// TIA Portal project "Project2" (V20)

(* hardware
DEVICE "S7-1200 station_1"  S7-1200 Station
   slot 0: "Rack_0"  S7-1200 Rack  Rack  V1.0
   slot 1: "PLC_1"  CPU 1214C DC/DC/DC  6ES7 214-1AG40-0XB0  V4.5
*)

// ===== PLC "PLC_1"  CPU 1214C DC/DC/DC =====

VAR_GLOBAL   // PLC tag table "Default tag table"
   "Axis_2_Pulse" AT %Q0.1 : Bool;
   "Axis_1_Direction" AT %Q0.6 : Bool;
   "Axis_Conveyor" AT %Q0.3 : Bool;
   "Axis_1_Pulse" AT %Q0.2 : Bool;
   "Axis_2_Direction" AT %Q0.4 : Bool;
   "M_Emergency" AT %M0.1 : Bool;
   "Velocity_1" AT %MD54 : Real;
   "Velocity_2" AT %MD58 : Real;
   "Velocity_3" AT %MD62 : Real;
   "I_Start" AT %I0.5 : Bool;
   "Set Velocity Conveyor" AT %MD80 : Real;
   "Velocity Conveyor" AT %MD84 : Real;
   "DeltaX_JobRev" AT %M200.1 : Bool;
   "DeltaX_JobFwd" AT %M200.0 : Bool;
   "DeltaX_Auto" AT %M11.0 : Bool;
   "EXC_Absolute" AT %M10.2 : Bool;
   "Po.S Done" AT %M120.0 : Bool;
   "Pos.DoneP" AT %M120.1 : Bool;
   "Servo#01 Fwd" AT %M2.0 : Bool;
   "Servo#02 Rev" AT %M2.1 : Bool;
   "Servo#02 Fwd" AT %M2.2 : Bool;
   "Servo#01 Rev" AT %M2.3 : Bool;
   "Servo#03 Fwd" AT %M2.4 : Bool;
   "Servo#03 Rev" AT %M2.5 : Bool;
   "Axis X_Work Complete" AT %M40.0 : Bool;
   "Axis Y_Work Complete" AT %M40.1 : Bool;
   "Axis Z_Work Complete" AT %M40.2 : Bool;
   "Axis X Busy" AT %M40.4 : Bool;
   "Axis Y Busy" AT %M40.5 : Bool;
   "Axis Z Busy" AT %M40.6 : Bool;
   "DeltaX_No Movement" AT %M40.7 : Bool;
   "I_Emergency" AT %I0.4 : Bool;
   "Vacum" AT %Q0.7 : Bool;
   "I_switch_1" AT %I0.0 : Bool;
   "DeltaX_Hbusy" AT %M111.0 : Bool;
   "DeltaX_Home" AT %M110.0 : Bool;
   "DeltaX_Start Home" AT %M110.1 : Bool;
   "tag_35" AT %M1000.0 : Bool;
   "I_switch_2" AT %I0.1 : Bool;
   "DeltaX1_1_Hbusy" AT %M111.1 : Bool;
   "Tag_39" AT %M1001.0 : Bool;
   "DeltaX2_Hbusy" AT %M111.2 : Bool;
   "DeltaX2_1_Hbusy" AT %M111.3 : Bool;
   "I_switch_3" AT %I0.2 : Bool;
   "Tag_40" AT %M1002.0 : Bool;
   "DeltaX3.1_Hbusy" AT %M111.5 : Bool;
   "DeltaX3_Hbusy" AT %M111.4 : Bool;
   "DeltaX_Home Busy" AT %M111.6 : Bool;
   "Home rest" AT %M110.2 : Bool;
   "EXC_Home P" AT %M152.0 : Bool;
   "Tag_28" AT %M305.1 : Bool;
   "ExC Home" AT %M150.7 : Bool;
   "Tag_27" AT %M305.0 : Bool;
   "Done_Home" AT %M10.3 : Bool;
   "Provess Data" AT %MW78 : Int;
   "Q_Reset_lamp" AT %Q8.5 : Bool;
   "PosionX_C#" AT %MD440 : Real;
   "PosionY_C#" AT %MD444 : Real;
   "Velocity_angular" AT %MD550 : Real;
   "DeltaX_Stop" AT %M11.1 : Bool;
   "bt_autoc#" AT %M110.3 : Bool;
   "bt_StopC#" AT %M110.4 : Bool;
   "DeltaX_Vacuum" AT %M153.0 : Bool;
   "Start Process" AT %M30.1 : Bool;
   "DeltaX_start Process" AT %M12.0 : Bool;
   "DeltaX_C# Enable" AT %M30.2 : Bool;
   "Tag_36" AT %M30.3 : Bool;
   "Step 7 ExC" AT %M151.1 : Bool;
   "Enable Scan" AT %M999.1 : Bool;
   "Tag_44" AT %M302.1 : Bool;
   "Tag_1" AT %M999.0 : Bool;
   "Step 1 Exc" AT %M150.0 : Bool;
   "Tag_2" AT %M140.7 : Bool;
   "PosX.Delta" AT %MD448 : Real;
   "PosY.Delta" AT %MD452 : Real;
   "Step 2 Exc" AT %M150.1 : Bool;
   "Step 3 Exc" AT %M150.2 : Bool;
   "Counter.PosX" AT %MD88 : Real;
   "Counter.PosY" AT %MD92 : Real;
   "Counter.PosZ" AT %MD96 : Real;
   "Step 4 Exc" AT %M150.3 : Bool;
   "Step 5 Exc" AT %M150.4 : Bool;
   "Counter.PosZ_1" AT %MD98 : Real;
   "Step 6 Exc" AT %M151.0 : Bool;
   "Tag_32" AT %M154.0 : Bool;
   "Tag_24" AT %M50.4 : Bool;
   "M#02 In" AT %M115.0 : Bool;
   "ExC" AT %M150.6 : Bool;
   "M#02 Out" AT %M115.1 : Bool;
   "DeltaX_Vaccum" AT %Q1.0 : Bool;
   "Tag_45" AT %M304.0 : Bool;
   "Tag_22" AT %Q1.1 : Bool;
   "M#02 Out Reset" AT %M115.2 : Bool;
   "M#02 StopSS" AT %I0.3 : Bool;
   "Tag_16" AT %MW4 : Word;
   "Tag_3" AT %M189.0 : Bool;
   "move_ss" AT %M45.0 : Bool;
   "Tag_4" AT %M45.1 : Bool;
   "EXC SS" AT %M158.0 : Bool;
   "EXC SS MOVE" AT %M158.1 : Bool;
   "Update_theta" AT %M700.0 : Bool;
   "Tag_6" AT %M700.1 : Bool;
   "Tag_7" AT %M700.2 : Bool;
   "m_theta1" AT %M121.0 : Bool;
   "Tag_5" AT %M121.1 : Bool;
   "m_theta2" AT %M121.2 : Bool;
   "Tag_9" AT %M121.3 : Bool;
   "m_theta3" AT %M121.4 : Bool;
   "Tag_10" AT %M121.5 : Bool;
   "move_ns" AT %M25.0 : Bool;
   "Tag_8" AT %M55.0 : Bool;
   "Tag_11" AT %MD100 : DInt;
   "Tag_12" AT %M56.0 : Bool;
   "Tag_13" AT %M57.0 : Bool;
   "Tag_14" AT %M152.1 : Bool;
   "move_abs" AT %M800.0 : Bool;
   "Home_c#" AT %M888.0 : Bool;
   "Tag_17" AT %M888.1 : Bool;
   "auto" AT %M880.0 : Bool;
   "SS" AT %M147.0 : Bool;
   "Tag_15" AT %M870.0 : Bool;
   "Tag_18" AT %M870.1 : Bool;
   "Tag_19" AT %M660.0 : Bool;
   "Tag_20" AT %M660.1 : Bool;
   "Tag_21" AT %M456.0 : Bool;
   "Tag_23" AT %M456.1 : Bool;
   "Tag_25" AT %MD6 : Real;
   "btn_auto" AT %M678.0 : Bool;
   "Tag_29" AT %M678.1 : Bool;
   "Tag_26" AT %M155.0 : Bool;
   "Tag_30" AT %M677.0 : Bool;
   "Tag_31" AT %MD14 : Real;
   "Tag_33" AT %MD15 : Real;
   "PosionZ_c#" AT %MD456 : Real;
   "Tag_34" AT %MD20 : Real;
   "Tag_37" AT %M78.0 : Bool;
   "Tag_38" AT %M78.1 : Bool;
   "Tag_41" AT %M78.2 : Bool;
   "Tag_42" AT %M88.0 : Bool;
   "Tag_43" AT %MD660 : DInt;
   "DeltaX_C# Enable_1" AT %M30.4 : Bool;
   "Tag_47" AT %M30.5 : Bool;
   "Servo1_Pulse" AT %Q0.0 : Bool;
   "Servo2_Direction" AT %Q0.5 : Bool;
   "Vitri_tha" AT %MW26 : Int;
   "DeltaX_C# Enable_2" AT %M30.6 : Bool;
   "Tag_48" AT %M30.7 : Bool;
   "DeltaX_C# Enable_3" AT %M31.0 : Bool;
   "Tag_49" AT %M31.1 : Bool;
   "DeltaX_C# Enable_4" AT %M31.2 : Bool;
   "Tag_50" AT %M31.3 : Bool;
   "DeltaX_C# Enable_5" AT %M31.4 : Bool;
   "Tag_51" AT %M31.5 : Bool;
   "Tag_46" AT %M37.0 : Bool;
   "Tag_52" AT %M37.1 : Bool;
   "Tag_53" AT %M37.2 : Bool;
   "Tag_54" AT %M37.3 : Bool;
   "Vat_1" AT %MD500 : DInt;
   "Vat_2" AT %MD504 : DInt;
   "Tag_55" AT %M37.4 : Bool;
   "Tag_56" AT %M37.5 : Bool;
   "Vat_3" AT %MD508 : DInt;
   "Tag_57" AT %M20.0 : Bool;
   "Tag_58" AT %M37.6 : Bool;
   "Tag_59" AT %M37.7 : Bool;
   "Tag_60" AT %M46.0 : Bool;
   "Tag_61" AT %M46.1 : Bool;
   "Tag_62" AT %M67.0 : Bool;
   "Tag_63" AT %M67.1 : Bool;
   "Tag_64" AT %MD50 : Real;
   "Delta_C# Enable_6" AT %M31.6 : Bool;
   "Delta_C# Enable_7" AT %M31.7 : Bool;
   "Delta_C# Enable_8" AT %M32.0 : Bool;
   "Delta_C# Enable_9" AT %M32.1 : Bool;
   "Delta_C# Enable_1.0" AT %M32.2 : Bool;
   "Delta_C# Enable_1.1" AT %M32.3 : Bool;
   "Delta_C# Enable_1.2" AT %M32.4 : Bool;
   "Delta_C# Enable_1.3" AT %M32.5 : Bool;
   "Delta_C# Enable_1.4" AT %M32.6 : Bool;
   "Tag_65" AT %M33.0 : Bool;
   "Tag_66" AT %M33.1 : Bool;
   "Tag_67" AT %M33.2 : Bool;
   "Tag_68" AT %M33.3 : Bool;
   "Tag_69" AT %M33.4 : Bool;
   "Tag_70" AT %M33.5 : Bool;
   "Tag_71" AT %M33.6 : Bool;
   "Tag_72" AT %M33.7 : Bool;
   "Tag_73" AT %M34.0 : Bool;
   "Tag_74" AT %M38.0 : Bool;
   "Tag_75" AT %M59.0 : Bool;
   "Tag_76" AT %M59.1 : Bool;
   "Tag_77" AT %M59.2 : Bool;
   "Tag_78" AT %M60.0 : Bool;
   "Tag_79" AT %M60.1 : Bool;
END_VAR

DATA_BLOCK "Position_Move_DB_3"   // DB10
{ S7_Optimized_Access := 'TRUE' }
VERSION : 0.1
// stored: InstanceOfName Position_Move
"Position_Move"
BEGIN
END_DATA_BLOCK

DATA_BLOCK "Singer_Inverse_Kinematics_Theta1"   // DB14
{ S7_Optimized_Access := 'TRUE' }
VERSION : 0.1
// stored: InstanceOfName Singer_Inverse_Kinematics
"Singer_Inverse_Kinematics"
BEGIN
END_DATA_BLOCK

DATA_BLOCK "Singer_Inverse_Kinematics_Theta2"   // DB15
{ S7_Optimized_Access := 'TRUE' }
VERSION : 0.1
// stored: InstanceOfName Singer_Inverse_Kinematics
"Singer_Inverse_Kinematics"
BEGIN
END_DATA_BLOCK

DATA_BLOCK "Singer_Inverse_Kinematics_Theta3"   // DB16
{ S7_Optimized_Access := 'TRUE' }
VERSION : 0.1
// stored: InstanceOfName Singer_Inverse_Kinematics
"Singer_Inverse_Kinematics"
BEGIN
END_DATA_BLOCK

DATA_BLOCK "Data_btn_vacum"   // DB17
{ S7_Optimized_Access := 'FALSE' }
VERSION : 0.1
   VAR
      btn_vacum_manual : Bool;
   END_VAR
BEGIN
END_DATA_BLOCK

DATA_BLOCK "Data_block_PLC_to_c#_NS"   // DB18
{ S7_Optimized_Access := 'FALSE' }
VERSION : 0.1
   VAR
      theta1 : Real;
      theta2 : Real;
      theta3 : Real;
      Busy : Bool;
      Done : Bool;
      Error : Bool;
   END_VAR
BEGIN
END_DATA_BLOCK

DATA_BLOCK "FC_Inverse_Kinematics_DB"   // DB20
{ S7_Optimized_Access := 'TRUE' }
VERSION : 0.1
// stored: InstanceOfName FB_Inverse_Kinematics
"FB_Inverse_Kinematics"
BEGIN
END_DATA_BLOCK

DATA_BLOCK "DB_CHECK_COORDINATION"   // DB31
{ S7_Optimized_Access := 'TRUE' }
VERSION : 0.1
   VAR
      Servo1_ss : Real;
      Servo2_ss : Real;
      Servo3_ss : Real;
      Z_Check : Real;
      X_Check_Ok : Real;
      X_Check : Real;
      Y_Check_Ok : Real;
      Z_Check_Ok : Real;
      theta_1_previous : Real;
      theta_2_previous : Real;
      theta_3_previous : Real;
      theta_1_check : Real;
      theta_2_check : Real;
      theta_3_check : Real;
      Y_Check : Real;
   END_VAR
BEGIN
END_DATA_BLOCK

DATA_BLOCK "Data_Button_C#_TO_PLC"   // DB33
{ S7_Optimized_Access := 'FALSE' }
VERSION : 0.1
   VAR
      btn_home : Bool;
   END_VAR
BEGIN
END_DATA_BLOCK

DATA_BLOCK "DB_Servo#01_PosC#"   // DB34
{ S7_Optimized_Access := 'FALSE' }
VERSION : 0.1
   VAR
      DataAxis_x : Real;
   END_VAR
BEGIN
END_DATA_BLOCK

DATA_BLOCK "DB_Servo#02_PosC#"   // DB35
{ S7_Optimized_Access := 'FALSE' }
VERSION : 0.1
   VAR
      DataAxis_Y : Real;
   END_VAR
BEGIN
END_DATA_BLOCK

DATA_BLOCK "DB_Servo#03_PosC#"   // DB36
{ S7_Optimized_Access := 'FALSE' }
VERSION : 0.1
   VAR
      DataAxis_Z : Real;
   END_VAR
BEGIN
END_DATA_BLOCK

DATA_BLOCK "KHOI_INVERSE_KINEMATIC_DB_1"   // DB37
{ S7_Optimized_Access := 'TRUE' }
VERSION : 0.1
// stored: InstanceOfName FB_Inverse_Kinematics
"FB_Inverse_Kinematics"
BEGIN
END_DATA_BLOCK

DATA_BLOCK "KHOI_INVERSE_KINEMATIC_DB"   // DB38
{ S7_Optimized_Access := 'TRUE' }
VERSION : 0.1
// stored: InstanceOfName FB_Inverse_Kinematics
"FB_Inverse_Kinematics"
BEGIN
END_DATA_BLOCK

DATA_BLOCK "DISTANT"   // DB39
{ S7_Optimized_Access := 'TRUE' }
VERSION : 0.1
   VAR
      TIME_DELAY_1 : Real;
      Y2 : Real;
      TIME_DELAY_2 : Real;
   END_VAR
BEGIN
END_DATA_BLOCK

DATA_BLOCK "Position_Move_DB"   // DB41
{ S7_Optimized_Access := 'TRUE' }
VERSION : 0.1
// stored: InstanceOfName Position_Move
"Position_Move"
BEGIN
END_DATA_BLOCK

DATA_BLOCK "Position_Move_DB_1"   // DB42
{ S7_Optimized_Access := 'TRUE' }
VERSION : 0.1
// stored: InstanceOfName Position_Move
"Position_Move"
BEGIN
END_DATA_BLOCK

DATA_BLOCK "Position_Move_DB_2"   // DB43
{ S7_Optimized_Access := 'TRUE' }
VERSION : 0.1
// stored: InstanceOfName Position_Move
"Position_Move"
BEGIN
END_DATA_BLOCK

DATA_BLOCK "Data_theta_c#_to_plc"   // DB44
{ S7_Optimized_Access := 'FALSE' }
VERSION : 0.1
   VAR
      theta1 : Real;
      theta2 : Real;
      theta3 : Real;
      velocity : Real;   // Set tốc độ từ C# xuống PLC
   END_VAR
BEGIN
END_DATA_BLOCK

DATA_BLOCK "Data_Emergency"   // DB45
{ S7_Optimized_Access := 'FALSE' }
VERSION : 0.1
   VAR
      s : Bool;
      btn_emergency : Bool := true;
   END_VAR
BEGIN
END_DATA_BLOCK

DATA_BLOCK "Data_Auto"   // DB46
{ S7_Optimized_Access := 'FALSE' }
VERSION : 0.1
   VAR
      btn_auto : Bool;
   END_VAR
BEGIN
END_DATA_BLOCK

DATA_BLOCK "Data_move_absolute"   // DB47
{ S7_Optimized_Access := 'FALSE' }
VERSION : 0.1
   VAR
      btn_move_abs : Bool;
   END_VAR
BEGIN
END_DATA_BLOCK

DATA_BLOCK "Data_rest"   // DB48
{ S7_Optimized_Access := 'FALSE' }
VERSION : 0.1
   VAR
      btn_rest : Bool;
   END_VAR
BEGIN
END_DATA_BLOCK

DATA_BLOCK "Data_Camera_toado"   // DB49
{ S7_Optimized_Access := 'FALSE' }
VERSION : 0.1
   VAR
      X : DInt;
      Y : DInt;
      Z : DInt;
      T : Int;
      "x+" : Real;
      "y+" : Real;
   END_VAR
BEGIN
END_DATA_BLOCK

DATA_BLOCK "Data_kiemtra_toado"   // DB50
{ S7_Optimized_Access := 'TRUE' }
VERSION : 0.1
   VAR
      x_convert : Real;
      y_convert : Real;
   END_VAR
BEGIN
END_DATA_BLOCK

DATA_BLOCK "Data_test"   // DB76
{ S7_Optimized_Access := 'FALSE' }
VERSION : 0.1
   VAR
      cos : Real;
      sin : Real;
   END_VAR
BEGIN
END_DATA_BLOCK

DATA_BLOCK "Data_Soluong_vat"   // DB77
{ S7_Optimized_Access := 'FALSE' }
VERSION : 0.1
   VAR
      Vat_1 : Real;
      Vat_2 : Real;
      Vat_3 : Real;
   END_VAR
BEGIN
END_DATA_BLOCK

DATA_BLOCK "Data_btn_start"   // DB78
{ S7_Optimized_Access := 'FALSE' }
VERSION : 0.1
   VAR
      Start : Bool;
   END_VAR
BEGIN
END_DATA_BLOCK

DATA_BLOCK "Data_Camera_c#_to_plc"   // DB80
{ S7_Optimized_Access := 'FALSE' }
VERSION : 0.1
   VAR
      x_camera : DInt;
      y_camera : DInt;
   END_VAR
BEGIN
END_DATA_BLOCK

DATA_BLOCK "data_btn_manual"   // DB81
{ S7_Optimized_Access := 'FALSE' }
VERSION : 0.1
   VAR
      btn_manual : Bool;
   END_VAR
BEGIN
END_DATA_BLOCK

DATA_BLOCK "Data_PLC_TO_C#_theta"   // DB111
{ S7_Optimized_Access := 'FALSE' }
VERSION : 0.1
   VAR
      Theta1 : Real;   // Đưa góc từ PLC lên C#
      Theta2 : Real;   // Đưa góc từ PLC lên C#
      Theta3 : Real;   // Đưa góc từ PLC lên C#
   END_VAR
BEGIN
END_DATA_BLOCK

// folder: System blocks/Program resources

DATA_BLOCK "RT_ready"   // DB30
{ S7_Optimized_Access := 'TRUE' }
AUTHOR : Simatic
FAMILY : IEC
NAME : IEC_TMR
VERSION : 1.0
// stored: InstanceOfName IEC_TIMER
"IEC_TIMER"
BEGIN
END_DATA_BLOCK

DATA_BLOCK "DeltaX_HomeDL"   // DB32
{ S7_Optimized_Access := 'TRUE' }
AUTHOR : Simatic
FAMILY : IEC
NAME : IEC_TMR
VERSION : 1.0
// stored: InstanceOfName IEC_TIMER
"IEC_TIMER"
BEGIN
END_DATA_BLOCK

DATA_BLOCK "IEC_Timer_0_DB"   // DB40
{ S7_Optimized_Access := 'TRUE' }
AUTHOR : Simatic
FAMILY : IEC
NAME : IEC_TMR
VERSION : 1.0
// stored: InstanceOfName IEC_TIMER
"IEC_TIMER"
BEGIN
END_DATA_BLOCK

DATA_BLOCK "IEC_Timer_0_DB_1"   // DB54
{ S7_Optimized_Access := 'TRUE' }
AUTHOR : Simatic
FAMILY : IEC
NAME : IEC_TMR
VERSION : 1.0
// stored: InstanceOfName IEC_TIMER
"IEC_TIMER"
BEGIN
END_DATA_BLOCK

DATA_BLOCK "01Step.DL"   // DB55
{ S7_Optimized_Access := 'TRUE' }
AUTHOR : Simatic
FAMILY : IEC
NAME : IEC_TMR
VERSION : 1.0
// stored: InstanceOfName IEC_TIMER
"IEC_TIMER"
BEGIN
END_DATA_BLOCK

DATA_BLOCK "IEC_Timer_0_DB_2"   // DB56
{ S7_Optimized_Access := 'TRUE' }
AUTHOR : Simatic
FAMILY : IEC
NAME : IEC_TMR
VERSION : 1.0
// stored: InstanceOfName IEC_TIMER
"IEC_TIMER"
BEGIN
END_DATA_BLOCK

DATA_BLOCK "02step.DL"   // DB57
{ S7_Optimized_Access := 'TRUE' }
AUTHOR : Simatic
FAMILY : IEC
NAME : IEC_TMR
VERSION : 1.0
// stored: InstanceOfName IEC_TIMER
"IEC_TIMER"
BEGIN
END_DATA_BLOCK

DATA_BLOCK "09step.DL"   // DB58
{ S7_Optimized_Access := 'TRUE' }
AUTHOR : Simatic
FAMILY : IEC
NAME : IEC_TMR
VERSION : 1.0
// stored: InstanceOfName IEC_TIMER
"IEC_TIMER"
BEGIN
END_DATA_BLOCK

DATA_BLOCK "VaccumDL"   // DB59
{ S7_Optimized_Access := 'TRUE' }
AUTHOR : Simatic
FAMILY : IEC
NAME : IEC_TMR
VERSION : 1.0
// stored: InstanceOfName IEC_TIMER
"IEC_TIMER"
BEGIN
END_DATA_BLOCK

DATA_BLOCK "IEC_Timer_0_DB_3"   // DB60
{ S7_Optimized_Access := 'TRUE' }
AUTHOR : Simatic
FAMILY : IEC
NAME : IEC_TMR
VERSION : 1.0
// stored: InstanceOfName IEC_TIMER
"IEC_TIMER"
BEGIN
END_DATA_BLOCK

DATA_BLOCK "03Step.DL"   // DB61
{ S7_Optimized_Access := 'TRUE' }
AUTHOR : Simatic
FAMILY : IEC
NAME : IEC_TMR
VERSION : 1.0
// stored: InstanceOfName IEC_TIMER
"IEC_TIMER"
BEGIN
END_DATA_BLOCK

DATA_BLOCK "IEC_Timer_0_DB_4"   // DB62
{ S7_Optimized_Access := 'TRUE' }
AUTHOR : Simatic
FAMILY : IEC
NAME : IEC_TMR
VERSION : 1.0
// stored: InstanceOfName IEC_TIMER
"IEC_TIMER"
BEGIN
END_DATA_BLOCK

DATA_BLOCK "#04Step.DL"   // DB63
{ S7_Optimized_Access := 'TRUE' }
AUTHOR : Simatic
FAMILY : IEC
NAME : IEC_TMR
VERSION : 1.0
// stored: InstanceOfName IEC_TIMER
"IEC_TIMER"
BEGIN
END_DATA_BLOCK

DATA_BLOCK "IEC_Timer_0_DB_5"   // DB64
{ S7_Optimized_Access := 'TRUE' }
AUTHOR : Simatic
FAMILY : IEC
NAME : IEC_TMR
VERSION : 1.0
// stored: InstanceOfName IEC_TIMER
"IEC_TIMER"
BEGIN
END_DATA_BLOCK

DATA_BLOCK "#05Step.DL"   // DB65
{ S7_Optimized_Access := 'TRUE' }
AUTHOR : Simatic
FAMILY : IEC
NAME : IEC_TMR
VERSION : 1.0
// stored: InstanceOfName IEC_TIMER
"IEC_TIMER"
BEGIN
END_DATA_BLOCK

DATA_BLOCK "IEC_Timer_0_DB_6"   // DB66
{ S7_Optimized_Access := 'TRUE' }
AUTHOR : Simatic
FAMILY : IEC
NAME : IEC_TMR
VERSION : 1.0
// stored: InstanceOfName IEC_TIMER
"IEC_TIMER"
BEGIN
END_DATA_BLOCK

DATA_BLOCK "#06Step.DL"   // DB67
{ S7_Optimized_Access := 'TRUE' }
AUTHOR : Simatic
FAMILY : IEC
NAME : IEC_TMR
VERSION : 1.0
// stored: InstanceOfName IEC_TIMER
"IEC_TIMER"
BEGIN
END_DATA_BLOCK

DATA_BLOCK "IEC_Timer_0_DB_7"   // DB68
{ S7_Optimized_Access := 'TRUE' }
AUTHOR : Simatic
FAMILY : IEC
NAME : IEC_TMR
VERSION : 1.0
// stored: InstanceOfName IEC_TIMER
"IEC_TIMER"
BEGIN
END_DATA_BLOCK

DATA_BLOCK "#07Step.DL"   // DB69
{ S7_Optimized_Access := 'TRUE' }
AUTHOR : Simatic
FAMILY : IEC
NAME : IEC_TMR
VERSION : 1.0
// stored: InstanceOfName IEC_TIMER
"IEC_TIMER"
BEGIN
END_DATA_BLOCK

DATA_BLOCK "IEC_Timer_0_DB_8"   // DB72
{ S7_Optimized_Access := 'TRUE' }
AUTHOR : Simatic
FAMILY : IEC
NAME : IEC_TMR
VERSION : 1.0
// stored: InstanceOfName IEC_TIMER
"IEC_TIMER"
BEGIN
END_DATA_BLOCK

// folder: (top level)

DATA_BLOCK "Servo2"   // DB1, Motion_DB
{ S7_Optimized_Access := 'TRUE' }
AUTHOR : SIMATIC
FAMILY : BasicMC
NAME : TO_PosAx
VERSION : 8.0
// stored: InstanceOfName TO_PositioningAxis
"TO_PositioningAxis"
BEGIN
   // Axis.OnlinePtoIndexCU = 1
   // Axis.HomingReferencePointSwitch_AddressCU = %I0.2
   // Axis.LengthUnitNormalized.Distance = 1005
   // Axis.DirectionOutputEnabledCU = TRUE
   // Axis.OnlinePtoModeCU = 16#0000_0002
   // Axis.SelectedChannel2EnumCU = %Q0.5
   // Axis.SelectedChannel1EnumCU = %Q0.1
   // Pulse.MinDeltaDeltaFrequencyCU = 0.004
   // Pulse.MaxDeltaDeltaFrequencyCU = 1.0E+10
   // Pulse.MinDeltaFrequencyCU = 0.005
   // Pulse.MaxDeltaFrequencyCU = 9.5E+9
   // Pulse.MinFrequencyCU = 1.0
   // Pulse.MaxFrequencyCU = 100000.0
   // Pulse.OutputSourceCU = 16#0000_0000
   // Axis.SelectPTO = 1
   // Axis.LengthUnit.LastDistance = 1005
END_DATA_BLOCK

DATA_BLOCK "Servo3"   // DB4, Motion_DB
{ S7_Optimized_Access := 'TRUE' }
AUTHOR : SIMATIC
FAMILY : BasicMC
NAME : TO_PosAx
VERSION : 8.0
// stored: InstanceOfName TO_PositioningAxis
"TO_PositioningAxis"
BEGIN
   // Axis.HomingReferencePointSwitch_AddressCU = %I0.1
   // Axis.LengthUnitNormalized.Distance = 1005
   // Axis.DirectionOutputEnabledCU = TRUE
   // Axis.OnlinePtoModeCU = 16#0000_0002
   // Axis.SelectedChannel2EnumCU = %Q0.6
   // Axis.SelectedChannel1EnumCU = %Q0.2
   // Pulse.MinDeltaDeltaFrequencyCU = 0.004
   // Pulse.MaxDeltaDeltaFrequencyCU = 1.0E+10
   // Pulse.MinDeltaFrequencyCU = 0.005
   // Pulse.MaxDeltaFrequencyCU = 9.5E+9
   // Pulse.MinFrequencyCU = 1.0
   // Pulse.MaxFrequencyCU = 100000.0
   // Pulse.OutputSourceCU = 16#0000_0000
   // Axis.SelectPTO = 2
   // Axis.OnlinePtoIndexCU = 2
   // Axis.LengthUnit.LastDistance = 1005
END_DATA_BLOCK

DATA_BLOCK "Servo1"   // DB5, Motion_DB
{ S7_Optimized_Access := 'TRUE' }
AUTHOR : SIMATIC
FAMILY : BasicMC
NAME : TO_PosAx
VERSION : 8.0
// stored: InstanceOfName TO_PositioningAxis
"TO_PositioningAxis"
BEGIN
   // Axis.HomingReferencePointSwitch_AddressCU = %I0.0
   // Axis.LengthUnitNormalized.Distance = 1005
   // Axis.DirectionOutputEnabledCU = TRUE
   // Axis.OnlinePtoModeCU = 16#0000_0002
   // Axis.SelectedChannel2EnumCU = %Q0.4
   // Axis.SelectedChannel1EnumCU = %Q0.0
   // Pulse.MinDeltaDeltaFrequencyCU = 0.004
   // Pulse.MaxDeltaDeltaFrequencyCU = 1.0E+10
   // Pulse.MinDeltaFrequencyCU = 0.005
   // Pulse.MaxDeltaFrequencyCU = 9.5E+9
   // Pulse.MinFrequencyCU = 1.0
   // Pulse.MaxFrequencyCU = 100000.0
   // Pulse.OutputSourceCU = 16#0000_0000
   // Axis.SelectPTO = 0
   // Axis.LengthUnit.LastDistance = 1005
END_DATA_BLOCK

DATA_BLOCK "Conveyor"   // DB19, Motion_DB
{ S7_Optimized_Access := 'TRUE' }
AUTHOR : SIMATIC
FAMILY : BasicMC
NAME : TO_PosAx
VERSION : 8.0
// stored: InstanceOfName TO_PositioningAxis
"TO_PositioningAxis"
BEGIN
   // Axis.OnlinePtoModeCU = 16#0000_0002
   // Axis.SelectedChannel2EnumCU = %Q0.7
   // Axis.SelectedChannel1EnumCU = %Q0.3
   // Pulse.MinDeltaDeltaFrequencyCU = 0.004
   // Pulse.MaxDeltaDeltaFrequencyCU = 1.0E+10
   // Pulse.MinDeltaFrequencyCU = 0.005
   // Pulse.MaxDeltaFrequencyCU = 9.5E+9
   // Pulse.MinFrequencyCU = 1.0
   // Pulse.MaxFrequencyCU = 100000.0
   // Pulse.OutputSourceCU = 16#0000_0000
   // Axis.SelectPTO = 3
   // Axis.OnlinePtoIndexCU = 3
   // Axis.LengthUnit.LastDistance = -1
END_DATA_BLOCK

FUNCTION_BLOCK "Singer_Inverse_Kinematics"   // FB1, LAD
{ S7_Optimized_Access := 'TRUE' }
VERSION : 0.1
   VAR_INPUT
      X : Real;
      Y : Real;
      Z : Real;
   END_VAR
   VAR_OUTPUT
      theta : Real;
   END_VAR
   VAR_TEMP
      Y1 : Real;
      Y0 : Real;
      "A" : Real;
      "B" : Real;
      D : Real;
      Yj : Real;
      Zj : Real;
      YY : Real;
      XX : Real;
   END_VAR
   VAR CONSTANT
      pi : Real := 3.141593;
      sqrt3 : Real := 1.732058;
      sin120 : Real := 0.8660254;
      cos120 : Real := -0.5;
      tan60 : Real := 1.732058;
      sin30 : Real := 0.5;
      tan30 : Real := 0.5773503;
      f : Real := 60.0;
      rf : Real := 150.0;
      "e" : Real := 40.0;
      re : Real := 310.0;
   END_VAR
BEGIN

REGION Network 1: tính A,B
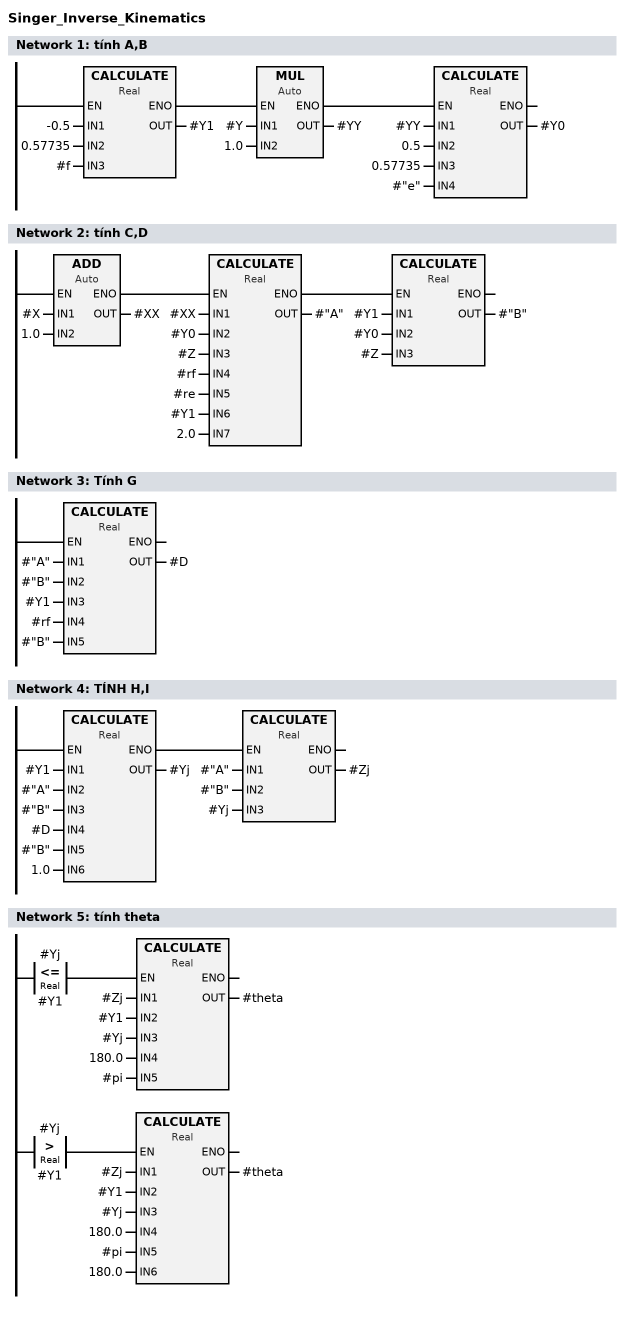
   RUNG wire#powerrail
      { S7_Templates := "SrcType := Real"; S7_Expression := "(IN1*IN2)*IN3" } Calculate(in1 := -0.5, in2 := 0.57735, in3 := #f, out => #Y1)
      Mul(in1 := #Y, in2 := 1.0, out => #YY)
      { S7_Templates := "SrcType := Real"; S7_Expression := "IN1-(IN2*IN3)*IN4" } Calculate(in1 := #YY, in2 := 0.5, in3 := 0.57735, in4 := #"e", out => #Y0)
   END_RUNG
   // the same network as SCL:
   #Y1 := ((-0.5)*0.57735)*#f;
   #YY := #Y * 1.0;
   #Y0 := #YY-(0.5*0.57735)*#"e";
END_REGION

REGION Network 2: tính C,D
   RUNG wire#powerrail
      Add(in1 := #X, in2 := 1.0, out => #XX)
      { S7_Templates := "SrcType := Real"; S7_Expression := "(IN1*IN1+IN2*IN2+IN3*IN3+IN4*IN4-IN5*IN5-IN6*IN6)/(IN7*IN3)" } Calculate(in1 := #XX, in2 := #Y0, in3 := #Z, in4 := #rf, in5 := #re, in6 := #Y1, in7 := 2.0, out => #"A")
      { S7_Templates := "SrcType := Real"; S7_Expression := "(IN1-IN2)/IN3" } Calculate(in1 := #Y1, in2 := #Y0, in3 := #Z, out => #"B")
   END_RUNG
   // the same network as SCL:
   #XX := #X + 1.0;
   #"A" := (#XX*#XX+#Y0*#Y0+#Z*#Z+#rf*#rf-#re*#re-#Y1*#Y1)/(2.0*#Z);
   #"B" := (#Y1-#Y0)/#Z;
END_REGION

REGION Network 3: Tính G
   RUNG wire#powerrail
      { S7_Templates := "SrcType := Real"; S7_Expression := "-(IN1+IN2*IN3)*(IN1+IN2*IN3)+IN4*(IN5*IN5*IN4+IN4)" } Calculate(in1 := #"A", in2 := #"B", in3 := #Y1, in4 := #rf, in5 := #"B", out => #D)
   END_RUNG
   // the same network as SCL:
   #D := -(#"A"+#"B"*#Y1)*(#"A"+#"B"*#Y1)+#rf*(#"B"*#"B"*#rf+#rf);
END_REGION

REGION Network 4: TÍNH H,I
   RUNG wire#powerrail
      { S7_Templates := "SrcType := Real"; S7_Expression := "(IN1-IN2*IN3-SQRT(IN4))/(IN5*IN5+IN6)" } Calculate(in1 := #Y1, in2 := #"A", in3 := #"B", in4 := #D, in5 := #"B", in6 := 1.0, out => #Yj)
      { S7_Templates := "SrcType := Real"; S7_Expression := "IN1+IN2*IN3" } Calculate(in1 := #"A", in2 := #"B", in3 := #Yj, out => #Zj)
   END_RUNG
   // the same network as SCL:
   #Yj := (#Y1-#"A"*#"B"-SQRT(#D))/(#"B"*#"B"+1.0);
   #Zj := #"A"+#"B"*#Yj;
END_REGION

REGION Network 5: tính theta
   RUNG wire#powerrail
      { S7_Templates := "SrcType := Real" } LE_Contact(in1 := #Yj, in2 := #Y1)
      { S7_Templates := "SrcType := Real"; S7_Expression := "ATAN(-IN1/(IN2-IN3))*IN4/IN5" } Calculate(in1 := #Zj, in2 := #Y1, in3 := #Yj, in4 := 180.0, in5 := #pi, out => #theta)
   END_RUNG
   RUNG wire#powerrail
      { S7_Templates := "SrcType := Real" } GT_Contact(in1 := #Yj, in2 := #Y1)
      { S7_Templates := "SrcType := Real"; S7_Expression := "ATAN(-IN1/(IN2-IN3))*IN4/IN5+IN6" } Calculate(in1 := #Zj, in2 := #Y1, in3 := #Yj, in4 := 180.0, in5 := #pi, in6 := 180.0, out => #theta)
   END_RUNG
   // the same network as SCL:
   IF #Yj <= #Y1 THEN #theta := ATAN(-#Zj/(#Y1-#Yj))*180.0/#pi; END_IF;
   IF #Yj > #Y1 THEN #theta := ATAN(-#Zj/(#Y1-#Yj))*180.0/#pi+180.0; END_IF;
END_REGION
END_FUNCTION_BLOCK

FUNCTION_BLOCK "FB_Inverse_Kinematics"   // FB2, LAD
{ S7_Optimized_Access := 'TRUE' }
VERSION : 0.1
   VAR_INPUT
      X0 : Real;
      Y0 : Real;
      Z0 : Real;
   END_VAR
   VAR_OUTPUT
      Theta1 : Real;
      Theta2 : Real;
      Theta3 : Real;
   END_VAR
   VAR_TEMP
      X1 : Real;
      Y1 : Real;
      X2 : Real;
      Y2 : Real;
   END_VAR
   VAR CONSTANT
      "-sin120" : Real := 0.8660254;
      cos120 : Real := -0.5;
   END_VAR
   VAR_TEMP   // added for the SCL form of the ladder/FBD networks
      _w1 : Bool;
      _w2 : Bool;
   END_VAR
BEGIN

REGION Network 1: Tính toán X,Y khi xoay 120 độ
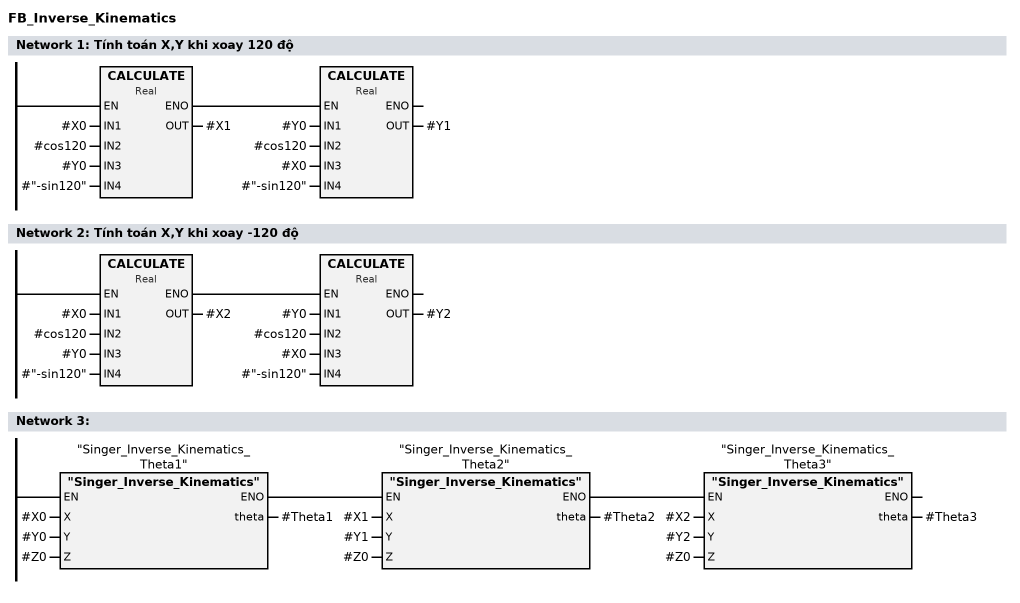
   RUNG wire#powerrail
      { S7_Templates := "SrcType := Real"; S7_Expression := "IN1*IN2+IN3*IN4" } Calculate(in1 := #X0, in2 := #cos120, in3 := #Y0, in4 := #"-sin120", out => #X1)
      { S7_Templates := "SrcType := Real"; S7_Expression := "IN1*IN2-IN3*IN4" } Calculate(in1 := #Y0, in2 := #cos120, in3 := #X0, in4 := #"-sin120", out => #Y1)
   END_RUNG
   // the same network as SCL:
   #X1 := #X0*#cos120+#Y0*#"-sin120";
   #Y1 := #Y0*#cos120-#X0*#"-sin120";
END_REGION

REGION Network 2: Tính toán X,Y khi xoay -120 độ
   RUNG wire#powerrail
      { S7_Templates := "SrcType := Real"; S7_Expression := "IN1*IN2-IN3*IN4" } Calculate(in1 := #X0, in2 := #cos120, in3 := #Y0, in4 := #"-sin120", out => #X2)
      { S7_Templates := "SrcType := Real"; S7_Expression := "IN1*IN2+IN3*IN4" } Calculate(in1 := #Y0, in2 := #cos120, in3 := #X0, in4 := #"-sin120", out => #Y2)
   END_RUNG
   // the same network as SCL:
   #X2 := #X0*#cos120-#Y0*#"-sin120";
   #Y2 := #Y0*#cos120+#X0*#"-sin120";
END_REGION

REGION Network 3
   RUNG wire#powerrail
      "Singer_Inverse_Kinematics_Theta1"(X := #X0, Y := #Y0, Z := #Z0, theta => #Theta1)
      "Singer_Inverse_Kinematics_Theta2"(X := #X1, Y := #Y1, Z := #Z0, theta => #Theta2)
      "Singer_Inverse_Kinematics_Theta3"(X := #X2, Y := #Y2, Z := #Z0, theta => #Theta3)
   END_RUNG
   // the same network as SCL:
   "Singer_Inverse_Kinematics_Theta1"(X := #X0, Y := #Y0, Z := #Z0, theta => #Theta1, ENO => #_w1);   // "Singer_Inverse_Kinematics"
   "Singer_Inverse_Kinematics_Theta2"(EN := #_w1, X := #X1, Y := #Y1, Z := #Z0, theta => #Theta2, ENO => #_w2);   // "Singer_Inverse_Kinematics"
   IF #_w2 THEN
       "Singer_Inverse_Kinematics_Theta3"(X := #X2, Y := #Y2, Z := #Z0, theta => #Theta3);   // "Singer_Inverse_Kinematics"
   END_IF;
END_REGION
END_FUNCTION_BLOCK

FUNCTION_BLOCK "Position_Move"   // FB3, LAD
{ S7_Optimized_Access := 'TRUE' }
VERSION : 0.1
   VAR_INPUT
      X_data : Real;
      Y_data : Real;
      Z_data : Real;
   END_VAR
BEGIN

REGION Network 1
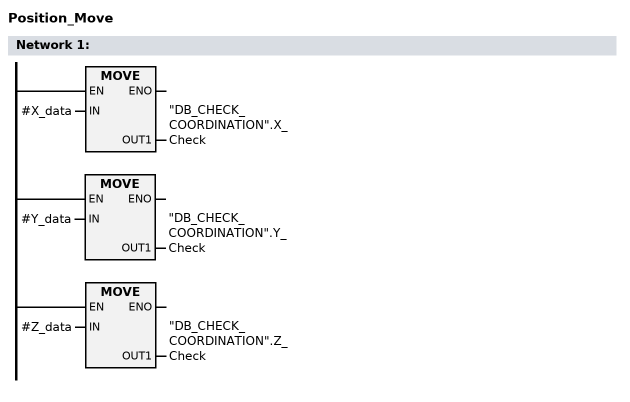
   RUNG wire#powerrail
      Move(in := #X_data, out1 => "DB_CHECK_COORDINATION".X_Check)
   END_RUNG
   RUNG wire#powerrail
      Move(in := #Y_data, out1 => "DB_CHECK_COORDINATION".Y_Check)
   END_RUNG
   RUNG wire#powerrail
      Move(in := #Z_data, out1 => "DB_CHECK_COORDINATION".Z_Check)
   END_RUNG
   // the same network as SCL:
   "DB_CHECK_COORDINATION".X_Check := #X_data;
   "DB_CHECK_COORDINATION".Y_Check := #Y_data;
   "DB_CHECK_COORDINATION".Z_Check := #Z_data;
END_REGION
END_FUNCTION_BLOCK

FUNCTION "FC_Axis" : Void   // FC1, LAD
{ S7_Optimized_Access := 'TRUE' }
VERSION : 0.1
   VAR_TEMP   // added for the SCL form of the ladder/FBD networks
      _w1 : Bool;
   END_VAR
BEGIN

REGION Network 1
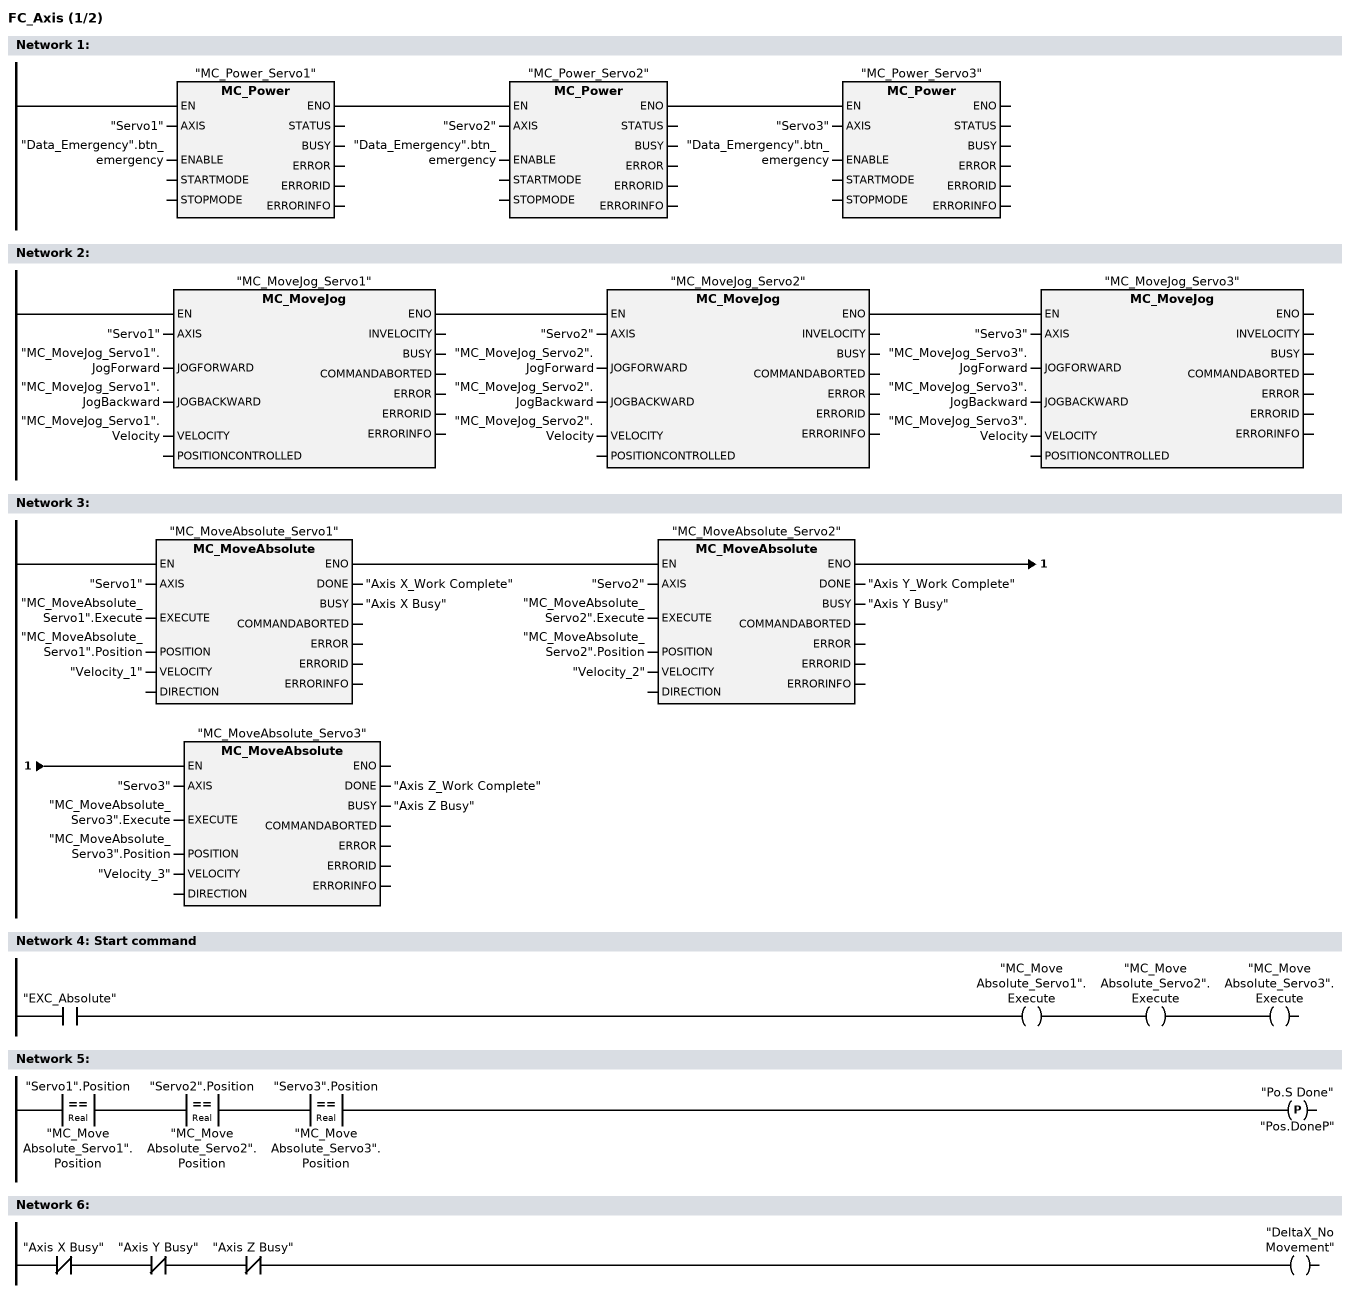
   // ENO of a box is taken as its EN; it also drops when the box reports an error
   "MC_Power_Servo1"(Axis := "Servo1", Enable := "Data_Emergency".btn_emergency);   // MC_Power
   "MC_Power_Servo2"(Axis := "Servo2", Enable := "Data_Emergency".btn_emergency);   // MC_Power
   "MC_Power_Servo3"(Axis := "Servo3", Enable := "Data_Emergency".btn_emergency);   // MC_Power
END_REGION

REGION Network 2
   // ENO of a box is taken as its EN; it also drops when the box reports an error
   "MC_MoveJog_Servo1"(Axis := "Servo1",   // MC_MoveJog
                       JogForward := "MC_MoveJog_Servo1".JogForward,
                       JogBackward := "MC_MoveJog_Servo1".JogBackward,
                       Velocity := "MC_MoveJog_Servo1".Velocity);
   "MC_MoveJog_Servo2"(Axis := "Servo2",   // MC_MoveJog
                       JogForward := "MC_MoveJog_Servo2".JogForward,
                       JogBackward := "MC_MoveJog_Servo2".JogBackward,
                       Velocity := "MC_MoveJog_Servo2".Velocity);
   "MC_MoveJog_Servo3"(Axis := "Servo3",   // MC_MoveJog
                       JogForward := "MC_MoveJog_Servo3".JogForward,
                       JogBackward := "MC_MoveJog_Servo3".JogBackward,
                       Velocity := "MC_MoveJog_Servo3".Velocity);
END_REGION

REGION Network 3
   // ENO of a box is taken as its EN; it also drops when the box reports an error
   "MC_MoveAbsolute_Servo1"(Axis := "Servo1",   // MC_MoveAbsolute
                           Execute := "MC_MoveAbsolute_Servo1".Execute,
                           Position := "MC_MoveAbsolute_Servo1".Position,
                           Velocity := "Velocity_1",
                           Done => "Axis X_Work Complete",
                           Busy => "Axis X Busy");
   "MC_MoveAbsolute_Servo2"(Axis := "Servo2",   // MC_MoveAbsolute
                           Execute := "MC_MoveAbsolute_Servo2".Execute,
                           Position := "MC_MoveAbsolute_Servo2".Position,
                           Velocity := "Velocity_2",
                           Done => "Axis Y_Work Complete",
                           Busy => "Axis Y Busy");
   "MC_MoveAbsolute_Servo3"(Axis := "Servo3",   // MC_MoveAbsolute
                           Execute := "MC_MoveAbsolute_Servo3".Execute,
                           Position := "MC_MoveAbsolute_Servo3".Position,
                           Velocity := "Velocity_3",
                           Done => "Axis Z_Work Complete",
                           Busy => "Axis Z Busy");
END_REGION

REGION Network 4: Start command
   RUNG wire#powerrail
      Contact( "EXC_Absolute" )
      Coil( "MC_MoveAbsolute_Servo1".Execute )
      Coil( "MC_MoveAbsolute_Servo2".Execute )
      Coil( "MC_MoveAbsolute_Servo3".Execute )
   END_RUNG
   // the same network as SCL:
   "MC_MoveAbsolute_Servo1".Execute := "EXC_Absolute";
   "MC_MoveAbsolute_Servo2".Execute := "EXC_Absolute";
   "MC_MoveAbsolute_Servo3".Execute := "EXC_Absolute";
END_REGION

REGION Network 5
   #_w1 := ("Servo1".Position = "MC_MoveAbsolute_Servo1".Position) AND ("Servo2".Position = "MC_MoveAbsolute_Servo2".Position) AND ("Servo3".Position = "MC_MoveAbsolute_Servo3".Position);
   "Po.S Done" := #_w1 AND NOT "Pos.DoneP";   // rising edge
   "Pos.DoneP" := #_w1;
END_REGION

REGION Network 6
   RUNG wire#powerrail
      I_Contact( "Axis X Busy" )
      I_Contact( "Axis Y Busy" )
      I_Contact( "Axis Z Busy" )
      Coil( "DeltaX_No Movement" )
   END_RUNG
   // the same network as SCL:
   "DeltaX_No Movement" := NOT "Axis X Busy" AND NOT "Axis Y Busy" AND NOT "Axis Z Busy";
END_REGION

REGION Network 7: Enable axis
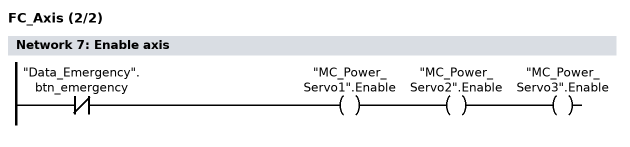
   RUNG wire#powerrail
      I_Contact( "Data_Emergency".btn_emergency )
      Coil( "MC_Power_Servo1".Enable )
      Coil( "MC_Power_Servo2".Enable )
      Coil( "MC_Power_Servo3".Enable )
   END_RUNG
   // the same network as SCL:
   "MC_Power_Servo1".Enable := NOT "Data_Emergency".btn_emergency;
   "MC_Power_Servo2".Enable := NOT "Data_Emergency".btn_emergency;
   "MC_Power_Servo3".Enable := NOT "Data_Emergency".btn_emergency;
END_REGION
END_FUNCTION

FUNCTION "FC_MOVE_Absolute" : Void   // FC3, LAD
{ S7_Optimized_Access := 'TRUE' }
VERSION : 0.1
BEGIN

REGION Network 1
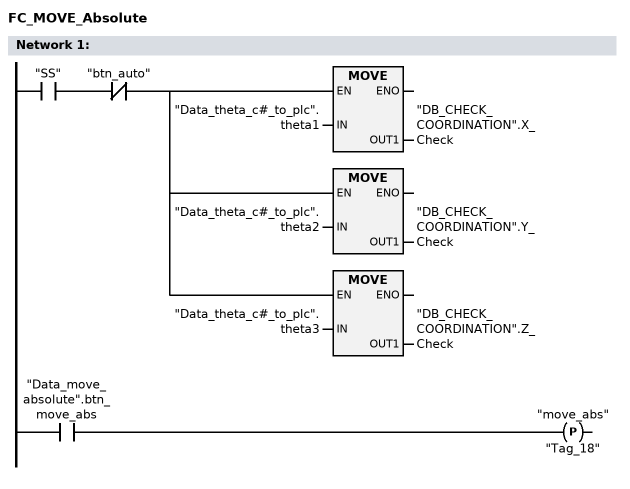
   IF "SS" AND NOT "btn_auto" THEN
       "DB_CHECK_COORDINATION".X_Check := "Data_theta_c#_to_plc".theta1;
       "DB_CHECK_COORDINATION".Y_Check := "Data_theta_c#_to_plc".theta2;
       "DB_CHECK_COORDINATION".Z_Check := "Data_theta_c#_to_plc".theta3;
   END_IF;
   "move_abs" := "Data_move_absolute".btn_move_abs AND NOT "Tag_18";   // rising edge
   "Tag_18" := "Data_move_absolute".btn_move_abs;
END_REGION
END_FUNCTION

FUNCTION "FC_Home" : Void   // FC4, LAD
{ S7_Optimized_Access := 'TRUE' }
VERSION : 0.1
   VAR_TEMP
      theta1_chuyendoi : Real;
      theta2_chuyendoi : Real;
      theta3_chuyendoi : Real;
   END_VAR
   VAR_TEMP   // added for the SCL form of the ladder/FBD networks
      _w1 : Bool;
      _w2 : Bool;
      _w3 : Bool;
   END_VAR
BEGIN

REGION Network 1
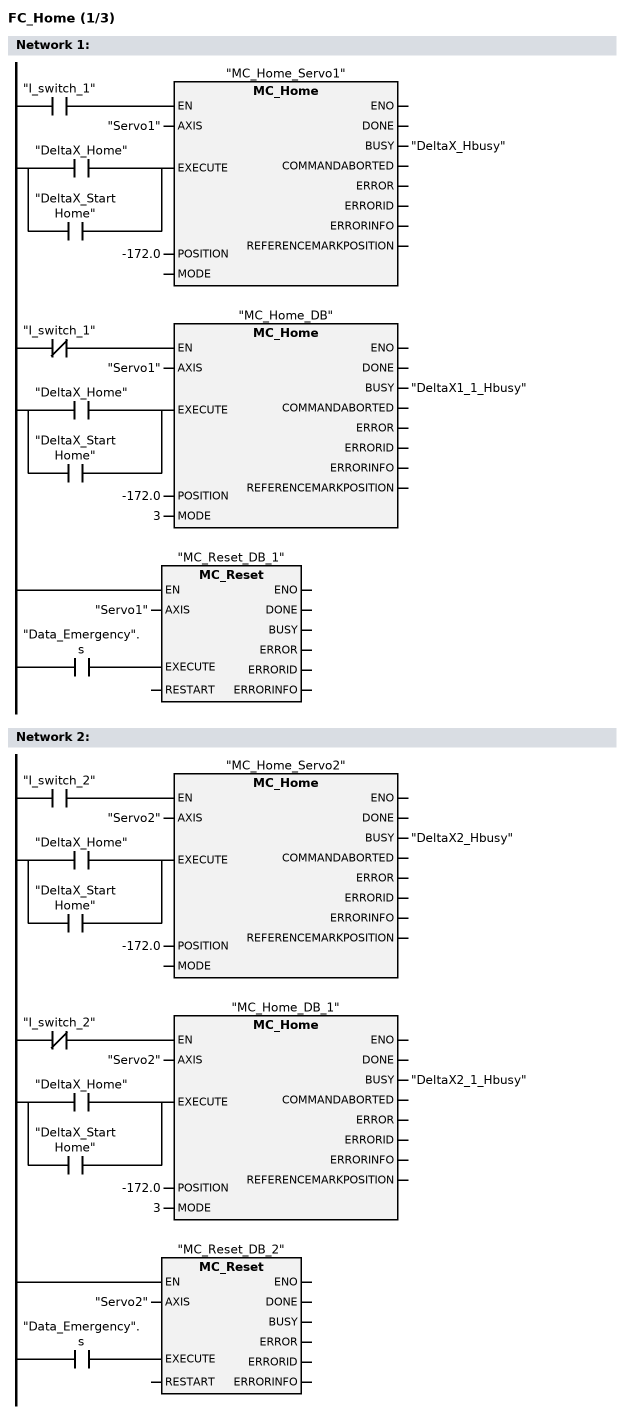
   IF "I_switch_1" THEN
       "MC_Home_Servo1"(Axis := "Servo1",   // MC_Home
                        Execute := "DeltaX_Home" OR "DeltaX_Start Home",
                        Position := -172.0,
                        Busy => "DeltaX_Hbusy");
   END_IF;
   IF NOT "I_switch_1" THEN
       "MC_Home_DB"(Axis := "Servo1",   // MC_Home
                    Execute := "DeltaX_Home" OR "DeltaX_Start Home",
                    Position := -172.0,
                    Mode := 3,
                    Busy => "DeltaX1_1_Hbusy");
   END_IF;
   "MC_Reset_DB_1"(Axis := "Servo1", Execute := "Data_Emergency".s);   // MC_Reset
END_REGION

REGION Network 2
   IF "I_switch_2" THEN
       "MC_Home_Servo2"(Axis := "Servo2",   // MC_Home
                        Execute := "DeltaX_Home" OR "DeltaX_Start Home",
                        Position := -172.0,
                        Busy => "DeltaX2_Hbusy");
   END_IF;
   IF NOT "I_switch_2" THEN
       "MC_Home_DB_1"(Axis := "Servo2",   // MC_Home
                      Execute := "DeltaX_Home" OR "DeltaX_Start Home",
                      Position := -172.0,
                      Mode := 3,
                      Busy => "DeltaX2_1_Hbusy");
   END_IF;
   "MC_Reset_DB_2"(Axis := "Servo2", Execute := "Data_Emergency".s);   // MC_Reset
END_REGION

REGION Network 3
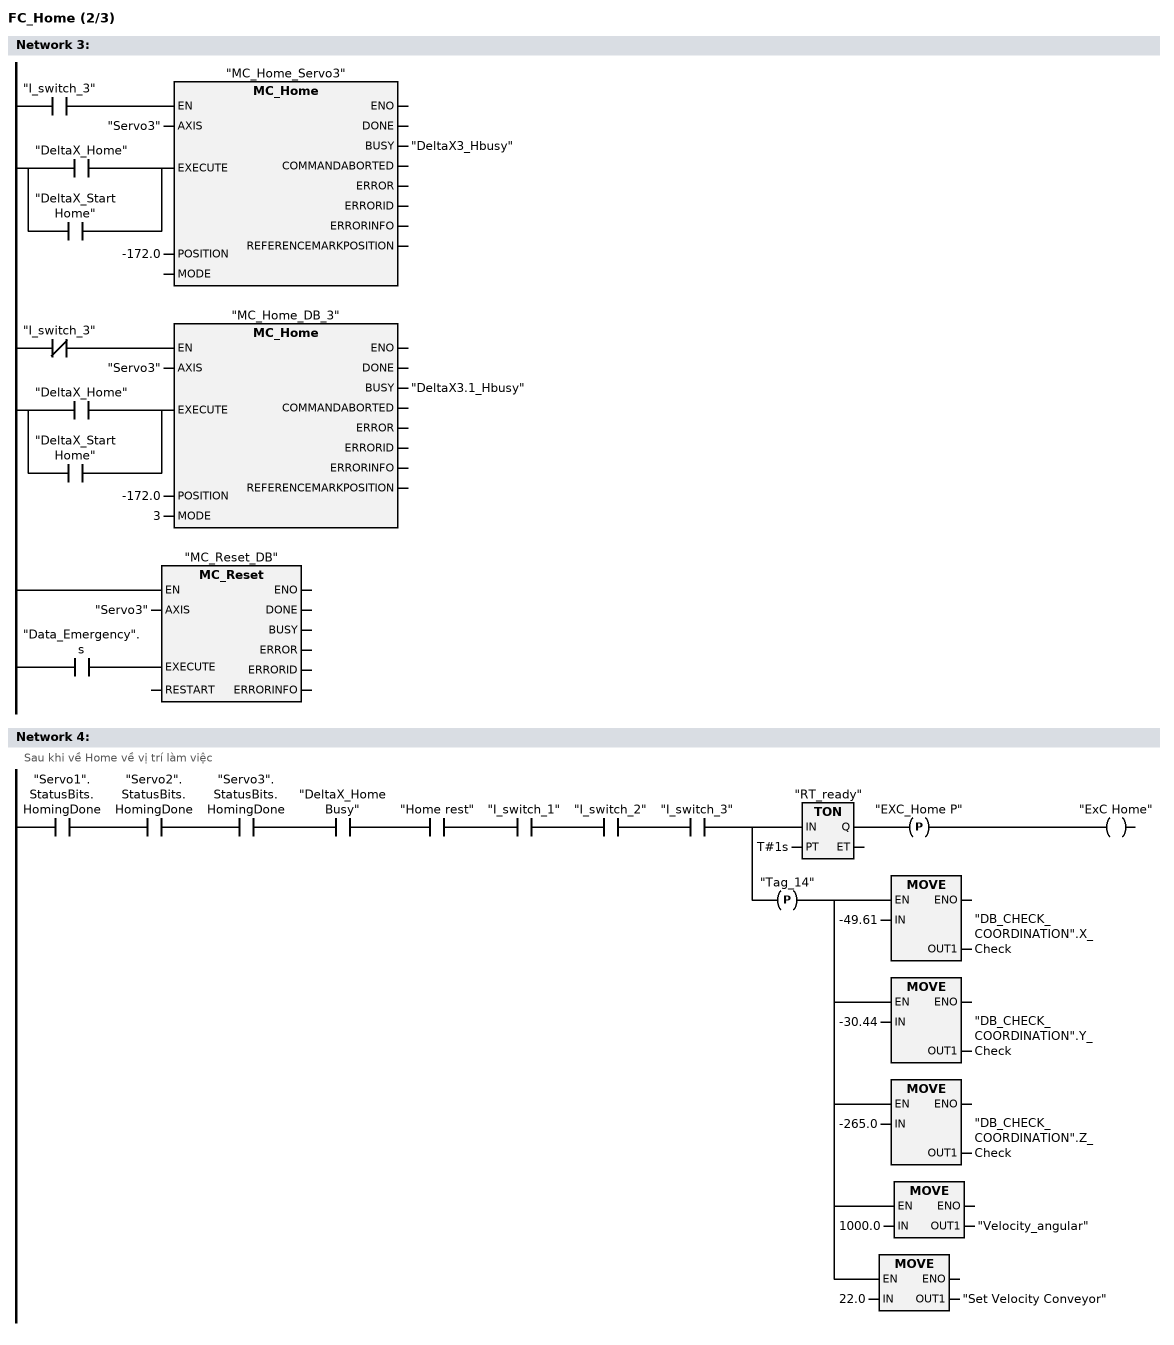
   IF "I_switch_3" THEN
       "MC_Home_Servo3"(Axis := "Servo3",   // MC_Home
                        Execute := "DeltaX_Home" OR "DeltaX_Start Home",
                        Position := -172.0,
                        Busy => "DeltaX3_Hbusy");
   END_IF;
   IF NOT "I_switch_3" THEN
       "MC_Home_DB_3"(Axis := "Servo3",   // MC_Home
                      Execute := "DeltaX_Home" OR "DeltaX_Start Home",
                      Position := -172.0,
                      Mode := 3,
                      Busy => "DeltaX3.1_Hbusy");
   END_IF;
   "MC_Reset_DB"(Axis := "Servo3", Execute := "Data_Emergency".s);   // MC_Reset
END_REGION

REGION Network 4
   // Sau khi về Home về vị trí làm việc
   #_w1 := "Servo1".StatusBits.HomingDone AND "Servo2".StatusBits.HomingDone AND "Servo3".StatusBits.HomingDone AND "DeltaX_Home Busy" AND "Home rest" AND "I_switch_1" AND "I_switch_2" AND "I_switch_3";
   "RT_ready".TON(IN := #_w1, PT := T#1s);
   #_w2 := "RT_ready".Q AND NOT "EXC_Home P";   // rising edge
   "EXC_Home P" := "RT_ready".Q;
   "ExC Home" := #_w2;
   #_w3 := #_w1 AND NOT "Tag_14";   // rising edge
   "Tag_14" := #_w1;
   IF #_w3 THEN
       "DB_CHECK_COORDINATION".X_Check := -49.61;
       "DB_CHECK_COORDINATION".Y_Check := -30.44;
       "DB_CHECK_COORDINATION".Z_Check := -265.0;
       "Velocity_angular" := 1000.0;
       "Set Velocity Conveyor" := 22.0;
   END_IF;
END_REGION

REGION Network 5
   // sau khi về home, thi cho phep san sang chay
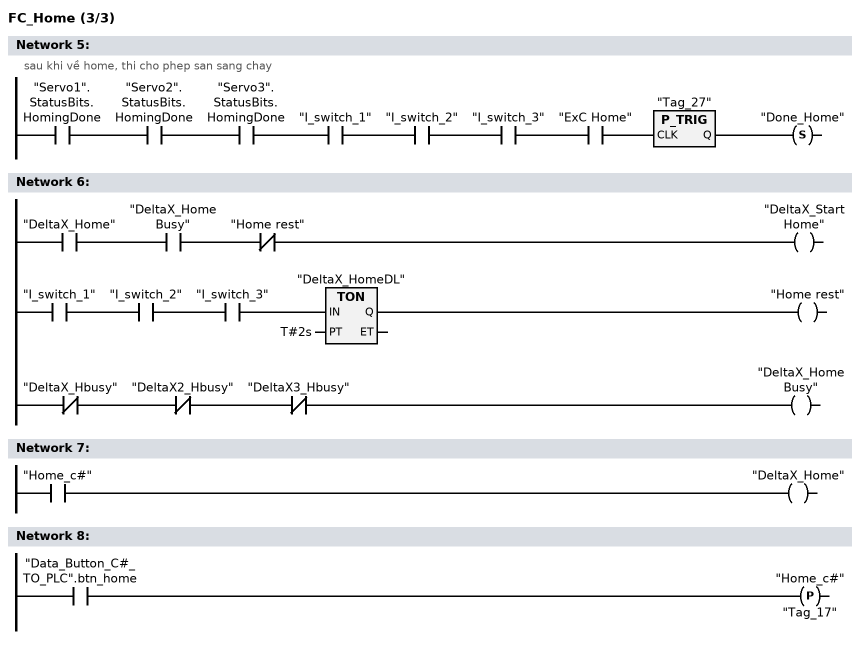
   RUNG wire#powerrail
      Contact( "Servo1".StatusBits.HomingDone )
      Contact( "Servo2".StatusBits.HomingDone )
      Contact( "Servo3".StatusBits.HomingDone )
      Contact( "I_switch_1" )
      Contact( "I_switch_2" )
      Contact( "I_switch_3" )
      Contact( "ExC Home" )
      P_Trig( "Tag_27" )
      S_Coil( "Done_Home" )
   END_RUNG
   // the same network as SCL:
   #_w1 := "Servo1".StatusBits.HomingDone AND "Servo2".StatusBits.HomingDone AND "Servo3".StatusBits.HomingDone AND "I_switch_1" AND "I_switch_2" AND "I_switch_3" AND "ExC Home";
   #_w2 := #_w1 AND NOT "Tag_27";   // rising edge
   "Tag_27" := #_w1;
   IF #_w2 THEN "Done_Home" := TRUE; END_IF;
END_REGION

REGION Network 6
   "DeltaX_Start Home" := "DeltaX_Home" AND "DeltaX_Home Busy" AND NOT "Home rest";
   "DeltaX_HomeDL".TON(IN := "I_switch_1" AND "I_switch_2" AND "I_switch_3", PT := T#2s);
   "Home rest" := "DeltaX_HomeDL".Q;
   "DeltaX_Home Busy" := NOT "DeltaX_Hbusy" AND NOT "DeltaX2_Hbusy" AND NOT "DeltaX3_Hbusy";
END_REGION

REGION Network 7
   RUNG wire#powerrail
      Contact( "Home_c#" )
      Coil( "DeltaX_Home" )
   END_RUNG
   // the same network as SCL:
   "DeltaX_Home" := "Home_c#";
END_REGION

REGION Network 8
   "Home_c#" := "Data_Button_C#_TO_PLC".btn_home AND NOT "Tag_17";   // rising edge
   "Tag_17" := "Data_Button_C#_TO_PLC".btn_home;
END_REGION
END_FUNCTION

FUNCTION "FC_Position" : Void   // FC5, LAD
{ S7_Optimized_Access := 'TRUE' }
VERSION : 0.1
BEGIN

REGION Network 1
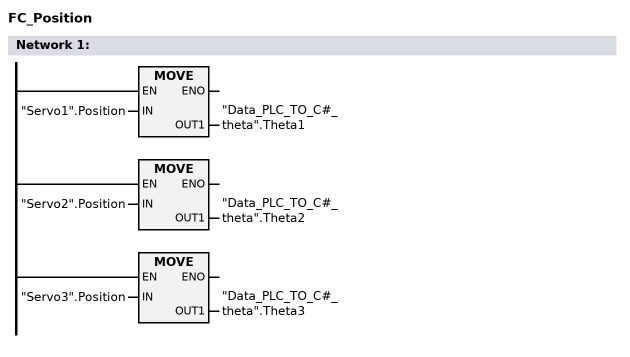
   RUNG wire#powerrail
      Move(in := "Servo1".Position, out1 => "Data_PLC_TO_C#_theta".Theta1)
   END_RUNG
   RUNG wire#powerrail
      Move(in := "Servo2".Position, out1 => "Data_PLC_TO_C#_theta".Theta2)
   END_RUNG
   RUNG wire#powerrail
      Move(in := "Servo3".Position, out1 => "Data_PLC_TO_C#_theta".Theta3)
   END_RUNG
   // the same network as SCL:
   "Data_PLC_TO_C#_theta".Theta1 := "Servo1".Position;
   "Data_PLC_TO_C#_theta".Theta2 := "Servo2".Position;
   "Data_PLC_TO_C#_theta".Theta3 := "Servo3".Position;
END_REGION
END_FUNCTION

FUNCTION "FC_Convert" : Void   // FC6, LAD
{ S7_Optimized_Access := 'TRUE' }
VERSION : 0.1
   VAR_INPUT
      theta_1 : Real;
      theta_2 : Real;
      theta_3 : Real;
   END_VAR
   VAR_OUTPUT
      theta_1_convert : Real;
      theta_2_convert : Real;
      theta_3_convert : Real;
   END_VAR
BEGIN

REGION Network 1
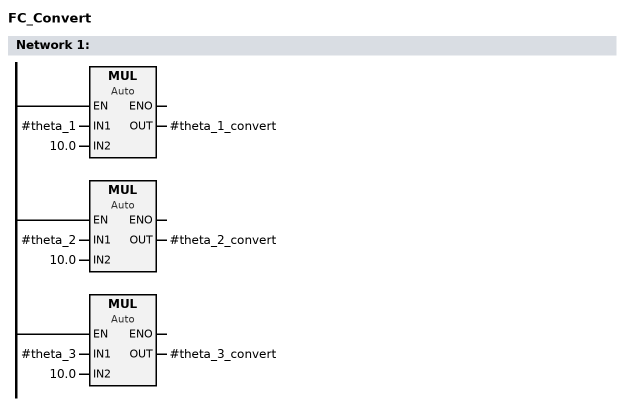
   RUNG wire#powerrail
      Mul(in1 := #theta_1, in2 := 10.0, out => #theta_1_convert)
   END_RUNG
   RUNG wire#powerrail
      Mul(in1 := #theta_2, in2 := 10.0, out => #theta_2_convert)
   END_RUNG
   RUNG wire#powerrail
      Mul(in1 := #theta_3, in2 := 10.0, out => #theta_3_convert)
   END_RUNG
   // the same network as SCL:
   #theta_1_convert := #theta_1 * 10.0;
   #theta_2_convert := #theta_2 * 10.0;
   #theta_3_convert := #theta_3 * 10.0;
END_REGION
END_FUNCTION

FUNCTION "FC_rest" : Void   // FC7, LAD
{ S7_Optimized_Access := 'TRUE' }
VERSION : 0.1
BEGIN

REGION Network 1
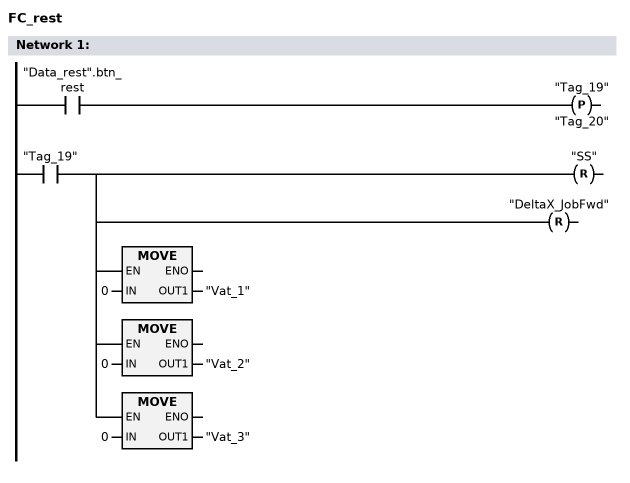
   "Tag_19" := "Data_rest".btn_rest AND NOT "Tag_20";   // rising edge
   "Tag_20" := "Data_rest".btn_rest;
   IF "Tag_19" THEN
       "SS" := FALSE;
       "DeltaX_JobFwd" := FALSE;
       "Vat_1" := 0;
       "Vat_2" := 0;
       "Vat_3" := 0;
   END_IF;
END_REGION
END_FUNCTION

FUNCTION "FC_Linmit_position" : Void   // FC8, LAD
{ S7_Optimized_Access := 'TRUE' }
VERSION : 0.1
   VAR_TEMP
      up_limit : Bool;
      R : Real;
      xy_limit : Bool;
      down_limit : Bool;
   END_VAR
BEGIN

REGION Network 1
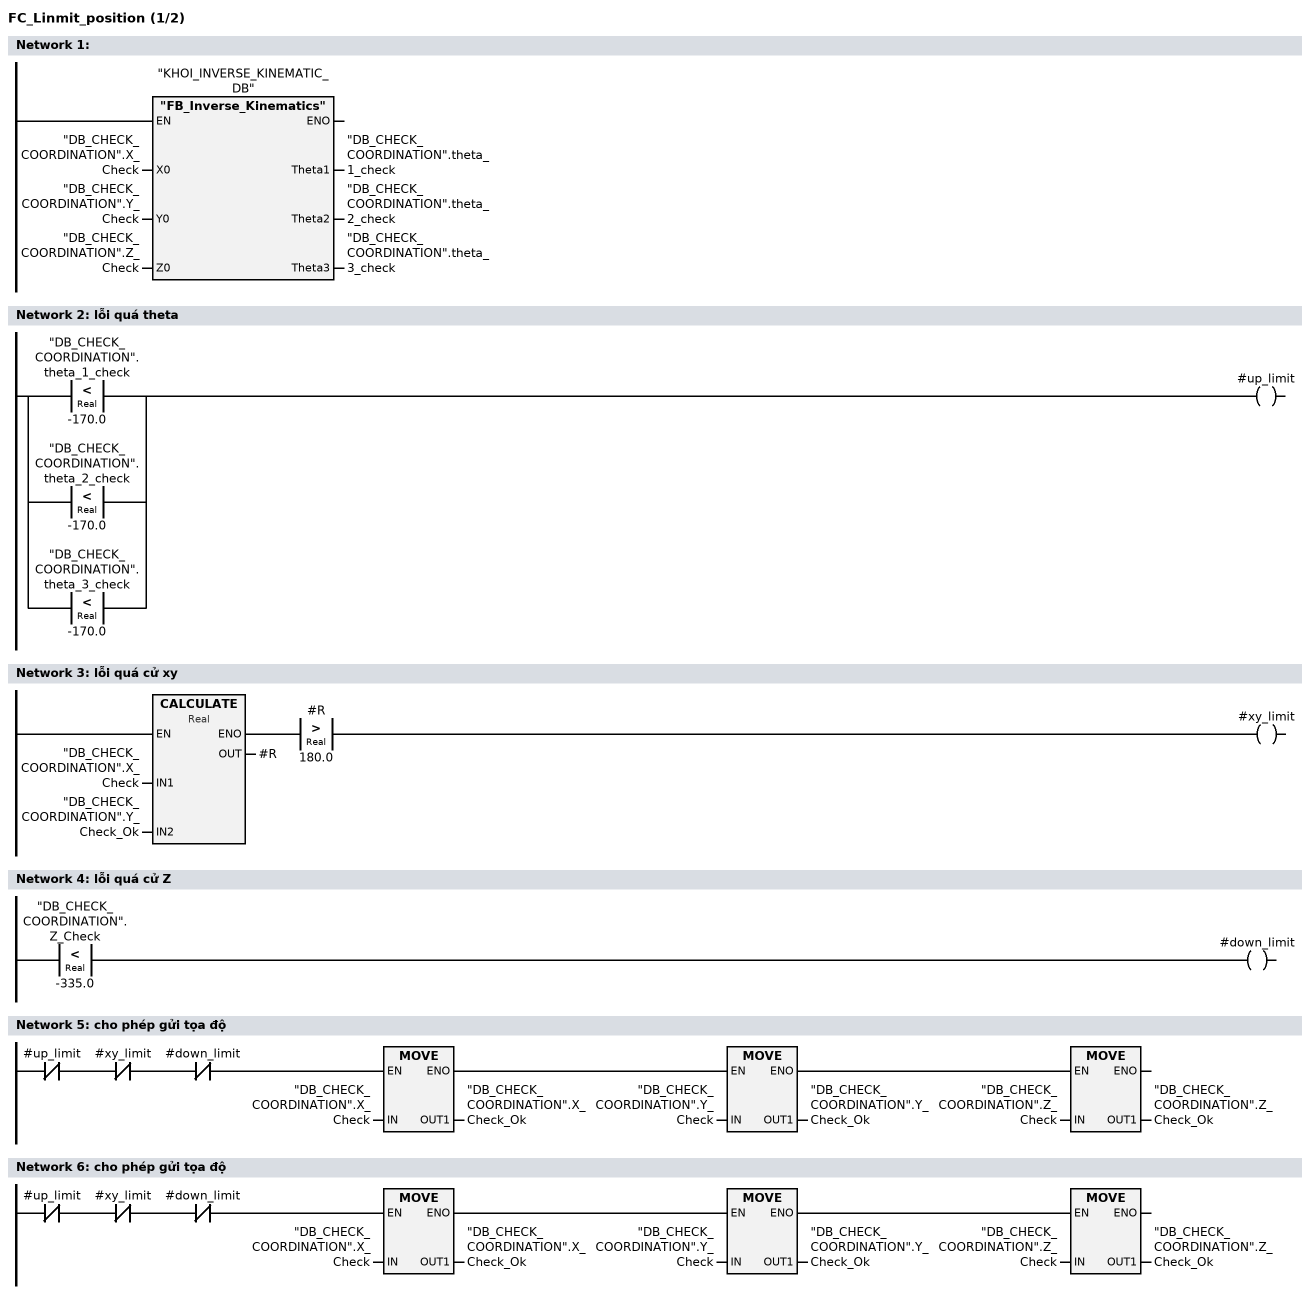
   RUNG wire#powerrail
      "KHOI_INVERSE_KINEMATIC_DB"(X0 := "DB_CHECK_COORDINATION".X_Check, Y0 := "DB_CHECK_COORDINATION".Y_Check, Z0 := "DB_CHECK_COORDINATION".Z_Check, Theta1 => "DB_CHECK_COORDINATION".theta_1_check, Theta2 => "DB_CHECK_COORDINATION".theta_2_check, Theta3 => "DB_CHECK_COORDINATION".theta_3_check)
   END_RUNG
   // the same network as SCL:
   "KHOI_INVERSE_KINEMATIC_DB"(X0 := "DB_CHECK_COORDINATION".X_Check,   // "FB_Inverse_Kinematics"
                           Y0 := "DB_CHECK_COORDINATION".Y_Check,
                           Z0 := "DB_CHECK_COORDINATION".Z_Check,
                           Theta1 => "DB_CHECK_COORDINATION".theta_1_check,
                           Theta2 => "DB_CHECK_COORDINATION".theta_2_check,
                           Theta3 => "DB_CHECK_COORDINATION".theta_3_check);
END_REGION

REGION Network 2: lỗi quá theta
   RUNG wire#powerrail
      { S7_Templates := "SrcType := Real" } LT_Contact(in1 := "DB_CHECK_COORDINATION".theta_1_check, in2 := -170.0)
      wire#w1
      Coil( #up_limit )
   END_RUNG
   RUNG wire#powerrail
      { S7_Templates := "SrcType := Real" } LT_Contact(in1 := "DB_CHECK_COORDINATION".theta_2_check, in2 := -170.0)
   END_RUNG wire#w1
   RUNG wire#powerrail
      { S7_Templates := "SrcType := Real" } LT_Contact(in1 := "DB_CHECK_COORDINATION".theta_3_check, in2 := -170.0)
   END_RUNG wire#w1
   // the same network as SCL:
   #up_limit := ("DB_CHECK_COORDINATION".theta_1_check < (-170.0)) OR ("DB_CHECK_COORDINATION".theta_2_check < (-170.0)) OR ("DB_CHECK_COORDINATION".theta_3_check < (-170.0));
END_REGION

REGION Network 3: lỗi quá cử xy
   RUNG wire#powerrail
      { S7_Templates := "SrcType := Real"; S7_Expression := "SQRT(IN1*IN1+IN2*IN2)" } Calculate(in1 := "DB_CHECK_COORDINATION".X_Check, in2 := "DB_CHECK_COORDINATION".Y_Check_Ok, out => #R)
      { S7_Templates := "SrcType := Real" } GT_Contact(in1 := #R, in2 := 180.0)
      Coil( #xy_limit )
   END_RUNG
   // the same network as SCL:
   #R := SQRT("DB_CHECK_COORDINATION".X_Check*"DB_CHECK_COORDINATION".X_Check+"DB_CHECK_COORDINATION".Y_Check_Ok*"DB_CHECK_COORDINATION".Y_Check_Ok);
   #xy_limit := #R > 180.0;
END_REGION

REGION Network 4: lỗi quá cử Z
   RUNG wire#powerrail
      { S7_Templates := "SrcType := Real" } LT_Contact(in1 := "DB_CHECK_COORDINATION".Z_Check, in2 := -335.0)
      Coil( #down_limit )
   END_RUNG
   // the same network as SCL:
   #down_limit := "DB_CHECK_COORDINATION".Z_Check < (-335.0);
END_REGION

REGION Network 5: cho phép gửi tọa độ
   RUNG wire#powerrail
      I_Contact( #up_limit )
      I_Contact( #xy_limit )
      I_Contact( #down_limit )
      Move(in := "DB_CHECK_COORDINATION".X_Check, out1 => "DB_CHECK_COORDINATION".X_Check_Ok)
      Move(in := "DB_CHECK_COORDINATION".Y_Check, out1 => "DB_CHECK_COORDINATION".Y_Check_Ok)
      Move(in := "DB_CHECK_COORDINATION".Z_Check, out1 => "DB_CHECK_COORDINATION".Z_Check_Ok)
   END_RUNG
   // the same network as SCL:
   IF NOT #up_limit AND NOT #xy_limit AND NOT #down_limit THEN
       "DB_CHECK_COORDINATION".X_Check_Ok := "DB_CHECK_COORDINATION".X_Check;
       "DB_CHECK_COORDINATION".Y_Check_Ok := "DB_CHECK_COORDINATION".Y_Check;
       "DB_CHECK_COORDINATION".Z_Check_Ok := "DB_CHECK_COORDINATION".Z_Check;
   END_IF;
END_REGION

REGION Network 6: cho phép gửi tọa độ
   RUNG wire#powerrail
      I_Contact( #up_limit )
      I_Contact( #xy_limit )
      I_Contact( #down_limit )
      Move(in := "DB_CHECK_COORDINATION".X_Check, out1 => "DB_CHECK_COORDINATION".X_Check_Ok)
      Move(in := "DB_CHECK_COORDINATION".Y_Check, out1 => "DB_CHECK_COORDINATION".Y_Check_Ok)
      Move(in := "DB_CHECK_COORDINATION".Z_Check, out1 => "DB_CHECK_COORDINATION".Z_Check_Ok)
   END_RUNG
   // the same network as SCL:
   IF NOT #up_limit AND NOT #xy_limit AND NOT #down_limit THEN
       "DB_CHECK_COORDINATION".X_Check_Ok := "DB_CHECK_COORDINATION".X_Check;
       "DB_CHECK_COORDINATION".Y_Check_Ok := "DB_CHECK_COORDINATION".Y_Check;
       "DB_CHECK_COORDINATION".Z_Check_Ok := "DB_CHECK_COORDINATION".Z_Check;
   END_IF;
END_REGION

REGION Network 7: đèn vàng báo lỗi
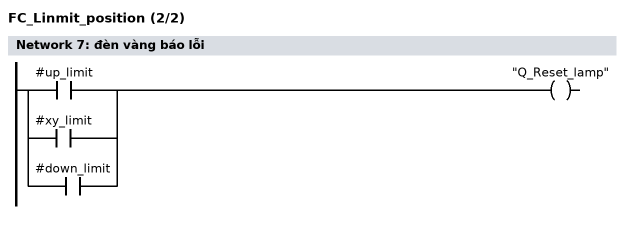
   RUNG wire#powerrail
      Contact( #up_limit )
      wire#w1
      Coil( "Q_Reset_lamp" )
   END_RUNG
   RUNG wire#powerrail
      Contact( #xy_limit )
   END_RUNG wire#w1
   RUNG wire#powerrail
      Contact( #down_limit )
   END_RUNG wire#w1
   // the same network as SCL:
   "Q_Reset_lamp" := #up_limit OR #xy_limit OR #down_limit;
END_REGION
END_FUNCTION

FUNCTION "FC_Conveyor" : Void   // FC10, LAD
{ S7_Optimized_Access := 'TRUE' }
VERSION : 0.1
BEGIN

REGION Network 1
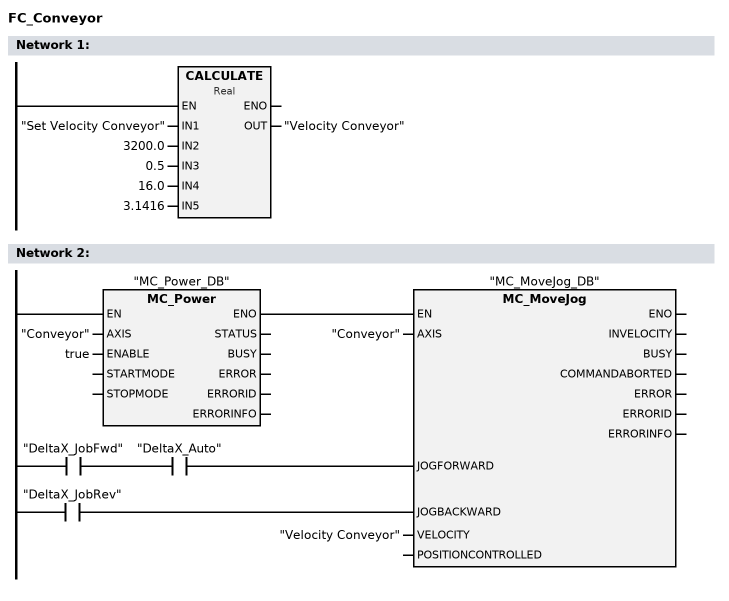
   RUNG wire#powerrail
      { S7_Templates := "SrcType := Real"; S7_Expression := "(IN1 * IN2) / (IN3 * (IN4 * IN5))" } Calculate(in1 := "Set Velocity Conveyor", in2 := 3200.0, in3 := 0.5, in4 := 16.0, in5 := 3.1416, out => "Velocity Conveyor")
   END_RUNG
   // the same network as SCL:
   "Velocity Conveyor" := ("Set Velocity Conveyor" * 3200.0) / (0.5 * (16.0 * 3.1416));
END_REGION

REGION Network 2
   // ENO of a box is taken as its EN; it also drops when the box reports an error
   "MC_Power_DB"(Axis := "Conveyor", Enable := true);   // MC_Power
   "MC_MoveJog_DB"(Axis := "Conveyor",   // MC_MoveJog
                   JogForward := "DeltaX_JobFwd" AND "DeltaX_Auto",
                   JogBackward := "DeltaX_JobRev",
                   Velocity := "Velocity Conveyor");
END_REGION
END_FUNCTION

FUNCTION "FC_Interpolation" : Void   // FC11, LAD
{ S7_Optimized_Access := 'TRUE' }
VERSION : 0.1
   VAR_INPUT
      Velcity_manual : Real;
   END_VAR
   VAR_OUTPUT
      Velocity_1 : Real;
      Velocity_2 : Real;
      Velocity_3 : Real;
   END_VAR
BEGIN

REGION Network 1
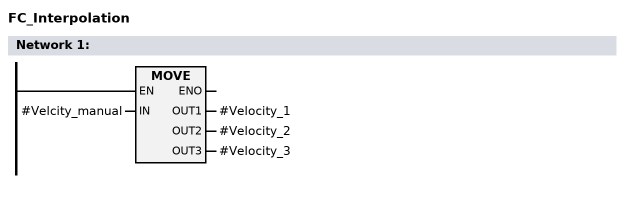
   RUNG wire#powerrail
      Move(in := #Velcity_manual, out1 => #Velocity_1, out2 => #Velocity_2, out3 => #Velocity_3)
   END_RUNG
   // the same network as SCL:
   #Velocity_1 := #Velcity_manual;
   #Velocity_2 := #Velcity_manual;
   #Velocity_3 := #Velcity_manual;
END_REGION
END_FUNCTION

FUNCTION "FC_Vacum" : Void   // FC12, LAD
{ S7_Optimized_Access := 'TRUE' }
VERSION : 0.1
BEGIN

REGION Network 1
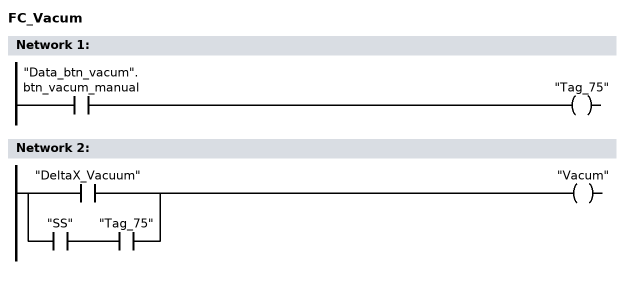
   RUNG wire#powerrail
      Contact( "Data_btn_vacum".btn_vacum_manual )
      Coil( "Tag_75" )
   END_RUNG
   // the same network as SCL:
   "Tag_75" := "Data_btn_vacum".btn_vacum_manual;
END_REGION

REGION Network 2
   RUNG wire#powerrail
      Contact( "DeltaX_Vacuum" )
      wire#w1
      Coil( "Vacum" )
   END_RUNG
   RUNG wire#powerrail
      Contact( "SS" )
      Contact( "Tag_75" )
   END_RUNG wire#w1
   // the same network as SCL:
   "Vacum" := "DeltaX_Vacuum" OR ("SS" AND "Tag_75");
END_REGION
END_FUNCTION

FUNCTION "FC_Auto" : Void   // FC13, LAD
{ S7_Optimized_Access := 'TRUE' }
VERSION : 0.1
   VAR_TEMP
      X_TT : Real;
      Y_TT : Real;
      Y_XD : Real;
      x_rotate : Real;
      y_rotate : Real;
      Vat_1 : DInt;
      Vat_2 : DInt;
      Vat_3 : DInt;
   END_VAR
   VAR CONSTANT
      "sin(150)" : Real := 0.5;
      "cos(150)" : Real := -0.866025;
   END_VAR
   VAR_TEMP   // added for the SCL form of the ladder/FBD networks
      _w1 : Bool;
      _w2 : Bool;
      _w3 : Bool;
      _w4 : Bool;
      _w5 : Bool;
      _w6 : Bool;
      _w7 : Bool;
      _w8 : Bool;
      _w9 : Bool;
      _w10 : Bool;
      _w11 : Bool;
      _w12 : Bool;
      _w13 : Bool;
      _w14 : Bool;
      _w15 : Bool;
   END_VAR
BEGIN

REGION Network 1
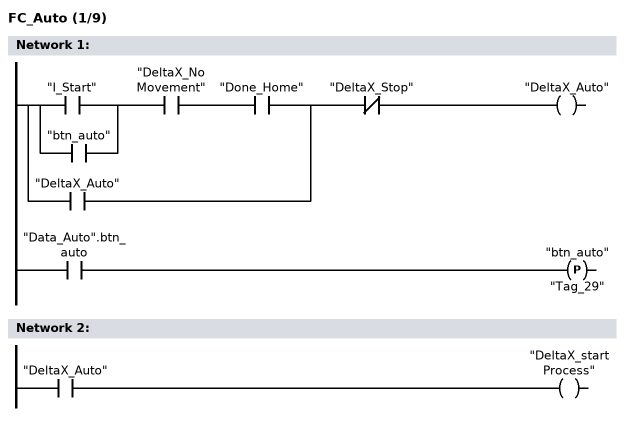
   "DeltaX_Auto" := ((("I_Start" OR "btn_auto") AND "DeltaX_No Movement" AND "Done_Home") OR "DeltaX_Auto") AND NOT "DeltaX_Stop";
   "btn_auto" := "Data_Auto".btn_auto AND NOT "Tag_29";   // rising edge
   "Tag_29" := "Data_Auto".btn_auto;
END_REGION

REGION Network 2
   RUNG wire#powerrail
      Contact( "DeltaX_Auto" )
      Coil( "DeltaX_start Process" )
   END_RUNG
   // the same network as SCL:
   "DeltaX_start Process" := "DeltaX_Auto";
END_REGION

REGION Network 3
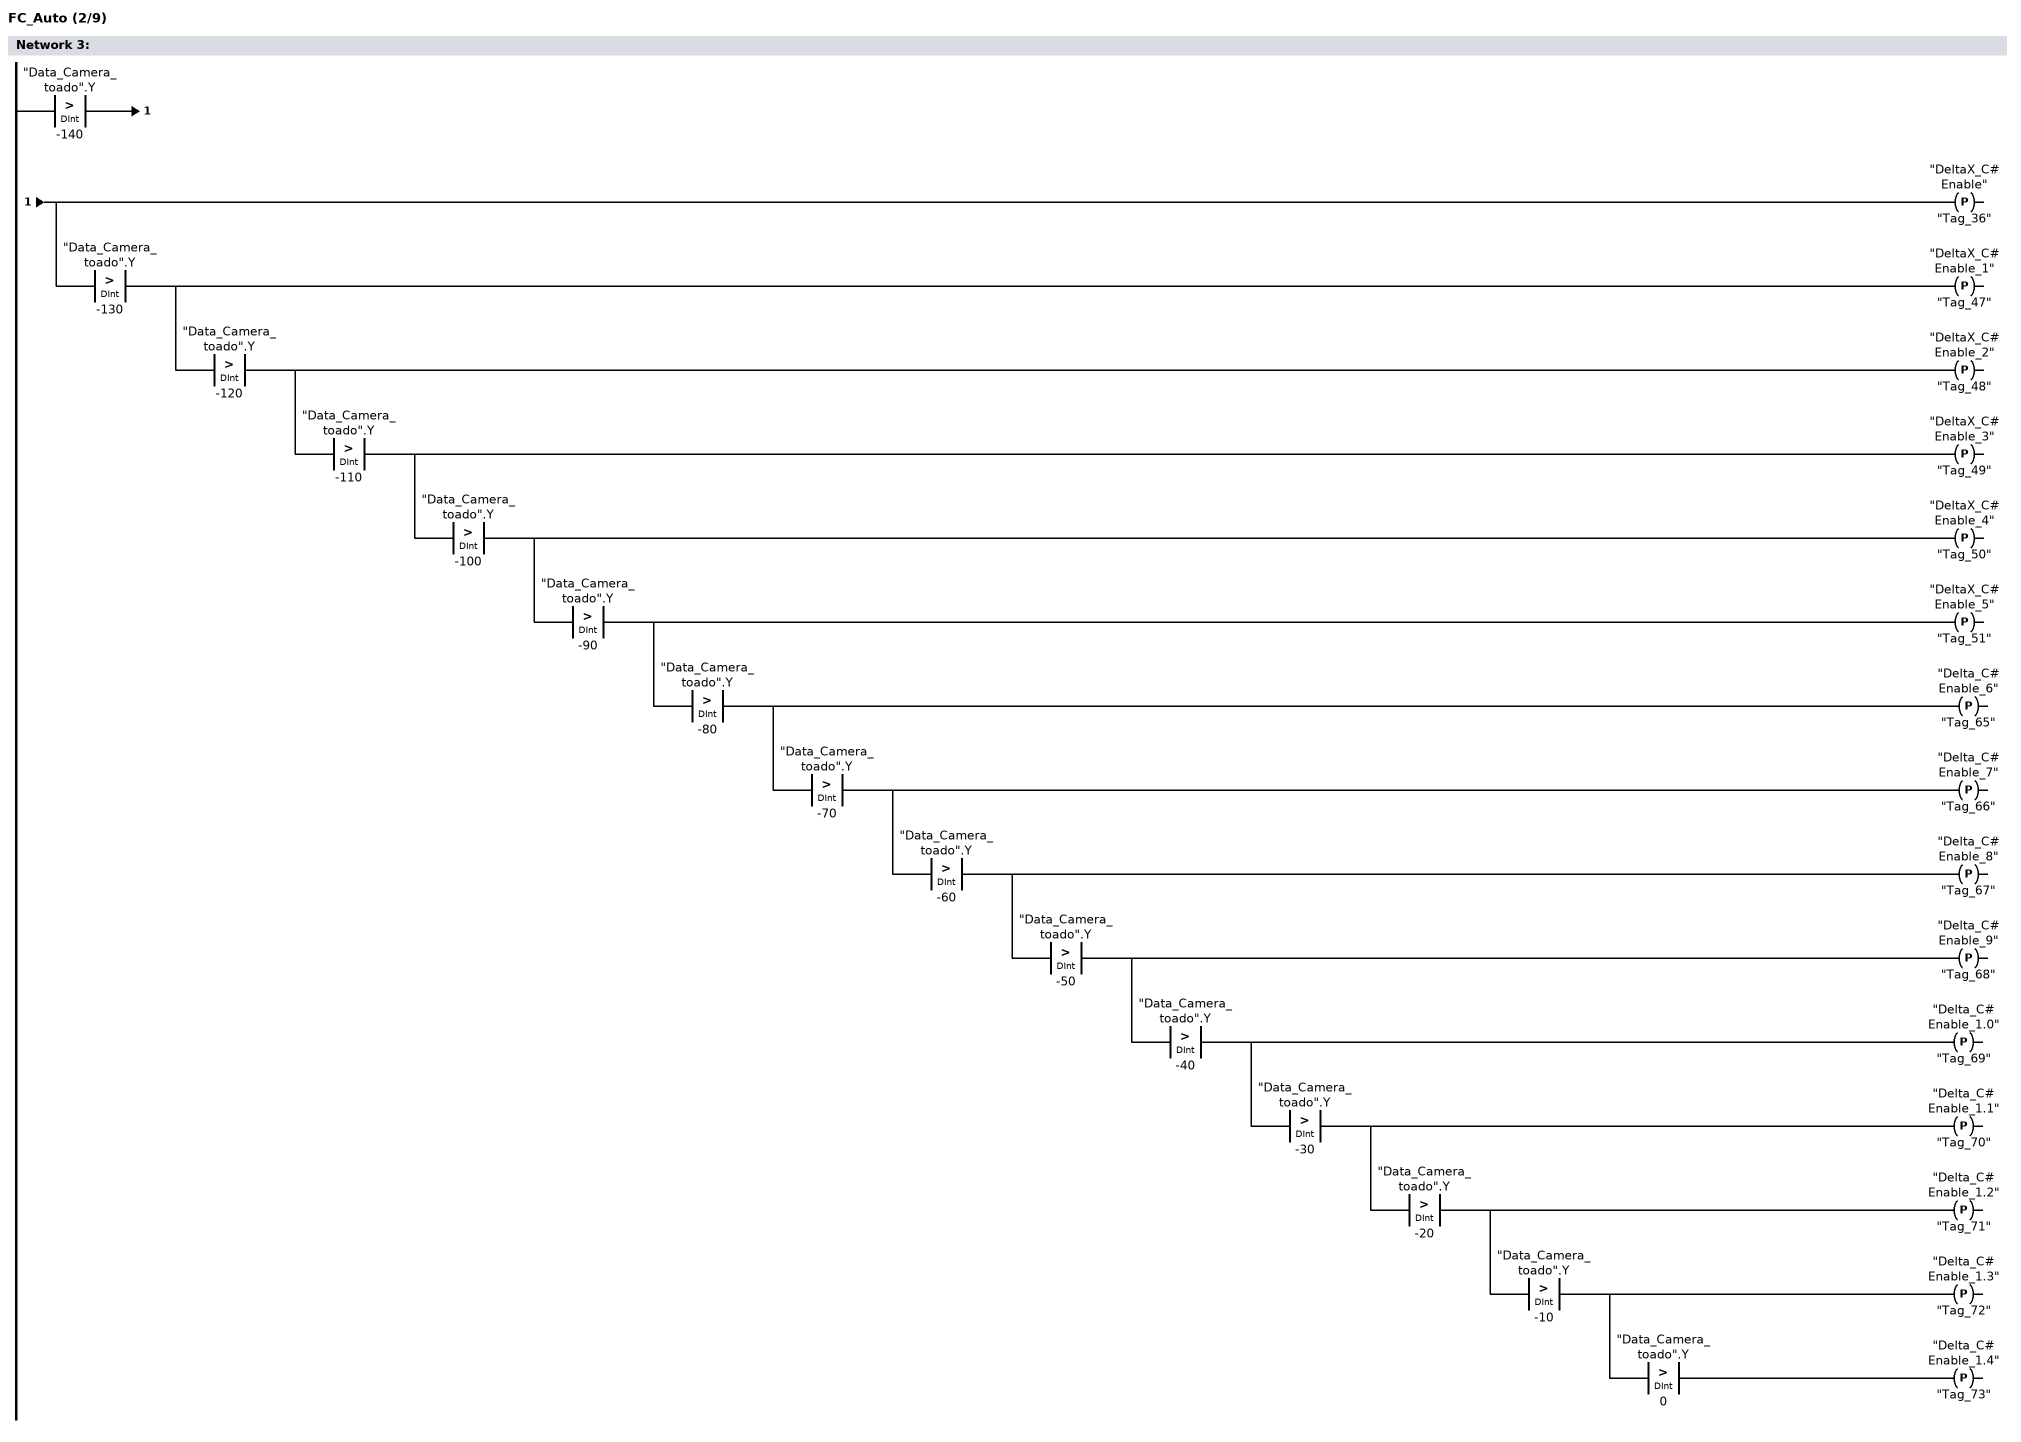
   #_w1 := "Data_Camera_toado".Y > (-140);
   "DeltaX_C# Enable" := #_w1 AND NOT "Tag_36";   // rising edge
   "Tag_36" := #_w1;
   #_w2 := #_w1 AND ("Data_Camera_toado".Y > (-130));
   "DeltaX_C# Enable_1" := #_w2 AND NOT "Tag_47";   // rising edge
   "Tag_47" := #_w2;
   #_w3 := #_w2 AND ("Data_Camera_toado".Y > (-120));
   "DeltaX_C# Enable_2" := #_w3 AND NOT "Tag_48";   // rising edge
   "Tag_48" := #_w3;
   #_w4 := #_w3 AND ("Data_Camera_toado".Y > (-110));
   "DeltaX_C# Enable_3" := #_w4 AND NOT "Tag_49";   // rising edge
   "Tag_49" := #_w4;
   #_w5 := #_w4 AND ("Data_Camera_toado".Y > (-100));
   "DeltaX_C# Enable_4" := #_w5 AND NOT "Tag_50";   // rising edge
   "Tag_50" := #_w5;
   #_w6 := #_w5 AND ("Data_Camera_toado".Y > (-90));
   "DeltaX_C# Enable_5" := #_w6 AND NOT "Tag_51";   // rising edge
   "Tag_51" := #_w6;
   #_w7 := #_w6 AND ("Data_Camera_toado".Y > (-80));
   "Delta_C# Enable_6" := #_w7 AND NOT "Tag_65";   // rising edge
   "Tag_65" := #_w7;
   #_w8 := #_w7 AND ("Data_Camera_toado".Y > (-70));
   "Delta_C# Enable_7" := #_w8 AND NOT "Tag_66";   // rising edge
   "Tag_66" := #_w8;
   #_w9 := #_w8 AND ("Data_Camera_toado".Y > (-60));
   "Delta_C# Enable_8" := #_w9 AND NOT "Tag_67";   // rising edge
   "Tag_67" := #_w9;
   #_w10 := #_w9 AND ("Data_Camera_toado".Y > (-50));
   "Delta_C# Enable_9" := #_w10 AND NOT "Tag_68";   // rising edge
   "Tag_68" := #_w10;
   #_w11 := #_w10 AND ("Data_Camera_toado".Y > (-40));
   "Delta_C# Enable_1.0" := #_w11 AND NOT "Tag_69";   // rising edge
   "Tag_69" := #_w11;
   #_w12 := #_w11 AND ("Data_Camera_toado".Y > (-30));
   "Delta_C# Enable_1.1" := #_w12 AND NOT "Tag_70";   // rising edge
   "Tag_70" := #_w12;
   #_w13 := #_w12 AND ("Data_Camera_toado".Y > (-20));
   "Delta_C# Enable_1.2" := #_w13 AND NOT "Tag_71";   // rising edge
   "Tag_71" := #_w13;
   #_w14 := #_w13 AND ("Data_Camera_toado".Y > (-10));
   "Delta_C# Enable_1.3" := #_w14 AND NOT "Tag_72";   // rising edge
   "Tag_72" := #_w14;
   #_w15 := #_w14 AND ("Data_Camera_toado".Y > 0);
   "Delta_C# Enable_1.4" := #_w15 AND NOT "Tag_73";   // rising edge
   "Tag_73" := #_w15;
END_REGION

REGION Network 4
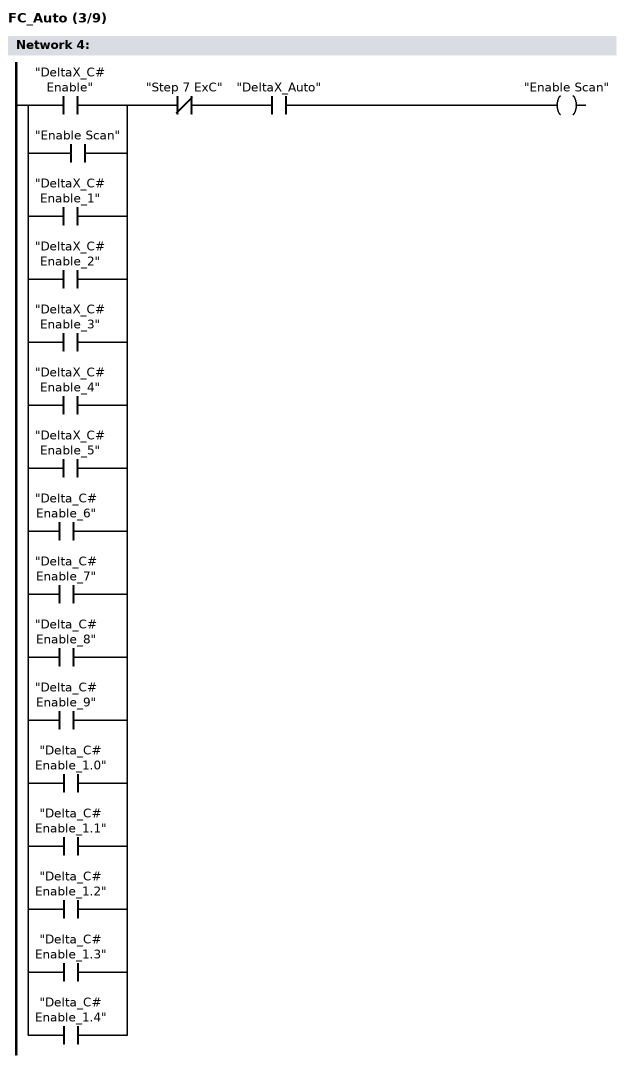
   RUNG wire#powerrail
      Contact( "DeltaX_C# Enable" )
      wire#w1
      I_Contact( "Step 7 ExC" )
      Contact( "DeltaX_Auto" )
      Coil( "Enable Scan" )
   END_RUNG
   RUNG wire#powerrail
      Contact( "Enable Scan" )
   END_RUNG wire#w1
   RUNG wire#powerrail
      Contact( "DeltaX_C# Enable_1" )
   END_RUNG wire#w1
   RUNG wire#powerrail
      Contact( "DeltaX_C# Enable_2" )
   END_RUNG wire#w1
   RUNG wire#powerrail
      Contact( "DeltaX_C# Enable_3" )
   END_RUNG wire#w1
   RUNG wire#powerrail
      Contact( "DeltaX_C# Enable_4" )
   END_RUNG wire#w1
   RUNG wire#powerrail
      Contact( "DeltaX_C# Enable_5" )
   END_RUNG wire#w1
   RUNG wire#powerrail
      Contact( "Delta_C# Enable_6" )
   END_RUNG wire#w1
   RUNG wire#powerrail
      Contact( "Delta_C# Enable_7" )
   END_RUNG wire#w1
   RUNG wire#powerrail
      Contact( "Delta_C# Enable_8" )
   END_RUNG wire#w1
   RUNG wire#powerrail
      Contact( "Delta_C# Enable_9" )
   END_RUNG wire#w1
   RUNG wire#powerrail
      Contact( "Delta_C# Enable_1.0" )
   END_RUNG wire#w1
   RUNG wire#powerrail
      Contact( "Delta_C# Enable_1.1" )
   END_RUNG wire#w1
   RUNG wire#powerrail
      Contact( "Delta_C# Enable_1.2" )
   END_RUNG wire#w1
   RUNG wire#powerrail
      Contact( "Delta_C# Enable_1.3" )
   END_RUNG wire#w1
   RUNG wire#powerrail
      Contact( "Delta_C# Enable_1.4" )
   END_RUNG wire#w1
   // the same network as SCL:
   "Enable Scan" := ("DeltaX_C# Enable" OR "Enable Scan" OR "DeltaX_C# Enable_1" OR "DeltaX_C# Enable_2" OR "DeltaX_C# Enable_3" OR "DeltaX_C# Enable_4" OR "DeltaX_C# Enable_5" OR "Delta_C# Enable_6" OR "Delta_C# Enable_7" OR "Delta_C# Enable_8" OR "Delta_C# Enable_9" OR "Delta_C# Enable_1.0" OR "Delta_C# Enable_1.1" OR "Delta_C# Enable_1.2" OR "Delta_C# Enable_1.3" OR "Delta_C# Enable_1.4") AND NOT "Step 7 ExC" AND "DeltaX_Auto";
END_REGION

REGION Network 5
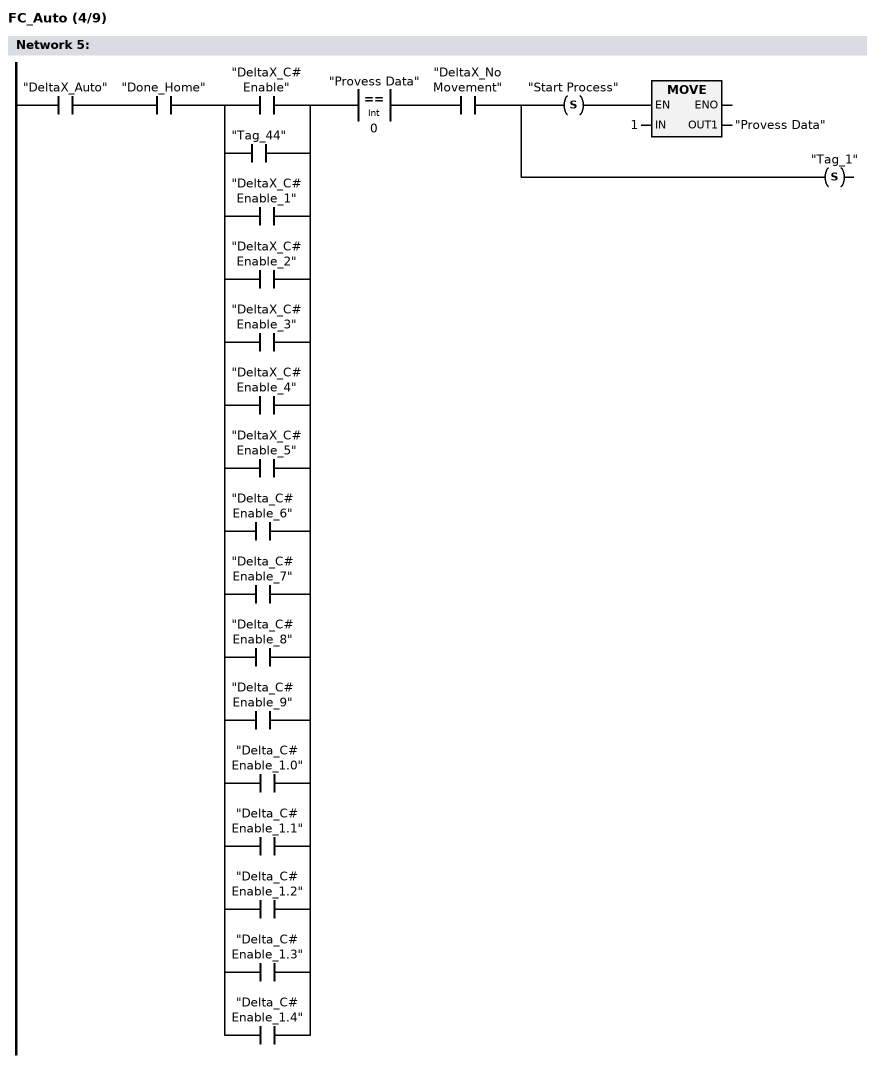
   RUNG wire#powerrail
      Contact( "DeltaX_Auto" )
      Contact( "Done_Home" )
      wire#w1
      Contact( "DeltaX_C# Enable" )
      wire#w2
      { S7_Templates := "SrcType := Int" } EQ_Contact(in1 := "Provess Data", in2 := 0)
      Contact( "DeltaX_No Movement" )
      wire#w3
      S_Coil( "Start Process" )
      Move(in := 1, out1 => "Provess Data")
   END_RUNG
   RUNG wire#w1
      Contact( "Tag_44" )
   END_RUNG wire#w2
   RUNG wire#w1
      Contact( "DeltaX_C# Enable_1" )
   END_RUNG wire#w2
   RUNG wire#w1
      Contact( "DeltaX_C# Enable_2" )
   END_RUNG wire#w2
   RUNG wire#w1
      Contact( "DeltaX_C# Enable_3" )
   END_RUNG wire#w2
   RUNG wire#w1
      Contact( "DeltaX_C# Enable_4" )
   END_RUNG wire#w2
   RUNG wire#w1
      Contact( "DeltaX_C# Enable_5" )
   END_RUNG wire#w2
   RUNG wire#w1
      Contact( "Delta_C# Enable_6" )
   END_RUNG wire#w2
   RUNG wire#w1
      Contact( "Delta_C# Enable_7" )
   END_RUNG wire#w2
   RUNG wire#w1
      Contact( "Delta_C# Enable_8" )
   END_RUNG wire#w2
   RUNG wire#w1
      Contact( "Delta_C# Enable_9" )
   END_RUNG wire#w2
   RUNG wire#w1
      Contact( "Delta_C# Enable_1.0" )
   END_RUNG wire#w2
   RUNG wire#w1
      Contact( "Delta_C# Enable_1.1" )
   END_RUNG wire#w2
   RUNG wire#w1
      Contact( "Delta_C# Enable_1.2" )
   END_RUNG wire#w2
   RUNG wire#w1
      Contact( "Delta_C# Enable_1.3" )
   END_RUNG wire#w2
   RUNG wire#w1
      Contact( "Delta_C# Enable_1.4" )
   END_RUNG wire#w2
   RUNG wire#w3
      S_Coil( "Tag_1" )
   END_RUNG
   // the same network as SCL:
   IF "DeltaX_Auto" AND "Done_Home" AND ("DeltaX_C# Enable" OR "Tag_44" OR "DeltaX_C# Enable_1" OR "DeltaX_C# Enable_2" OR "DeltaX_C# Enable_3" OR "DeltaX_C# Enable_4" OR "DeltaX_C# Enable_5" OR "Delta_C# Enable_6" OR "Delta_C# Enable_7" OR "Delta_C# Enable_8" OR "Delta_C# Enable_9" OR "Delta_C# Enable_1.0" OR "Delta_C# Enable_1.1" OR "Delta_C# Enable_1.2" OR "Delta_C# Enable_1.3" OR "Delta_C# Enable_1.4") AND ("Provess Data" = 0) AND "DeltaX_No Movement" THEN
       "Start Process" := TRUE;
   END_IF;
   #_w1 := "DeltaX_Auto" AND "Done_Home" AND ("DeltaX_C# Enable" OR "Tag_44" OR "DeltaX_C# Enable_1" OR "DeltaX_C# Enable_2" OR "DeltaX_C# Enable_3" OR "DeltaX_C# Enable_4" OR "DeltaX_C# Enable_5" OR "Delta_C# Enable_6" OR "Delta_C# Enable_7" OR "Delta_C# Enable_8" OR "Delta_C# Enable_9" OR "Delta_C# Enable_1.0" OR "Delta_C# Enable_1.1" OR "Delta_C# Enable_1.2" OR "Delta_C# Enable_1.3" OR "Delta_C# Enable_1.4") AND ("Provess Data" = 0) AND "DeltaX_No Movement";
   IF #_w1 THEN
       "Provess Data" := 1;
       "Tag_1" := TRUE;
   END_IF;
END_REGION

REGION Network 6: DI chuyển xy đến vị trí vật
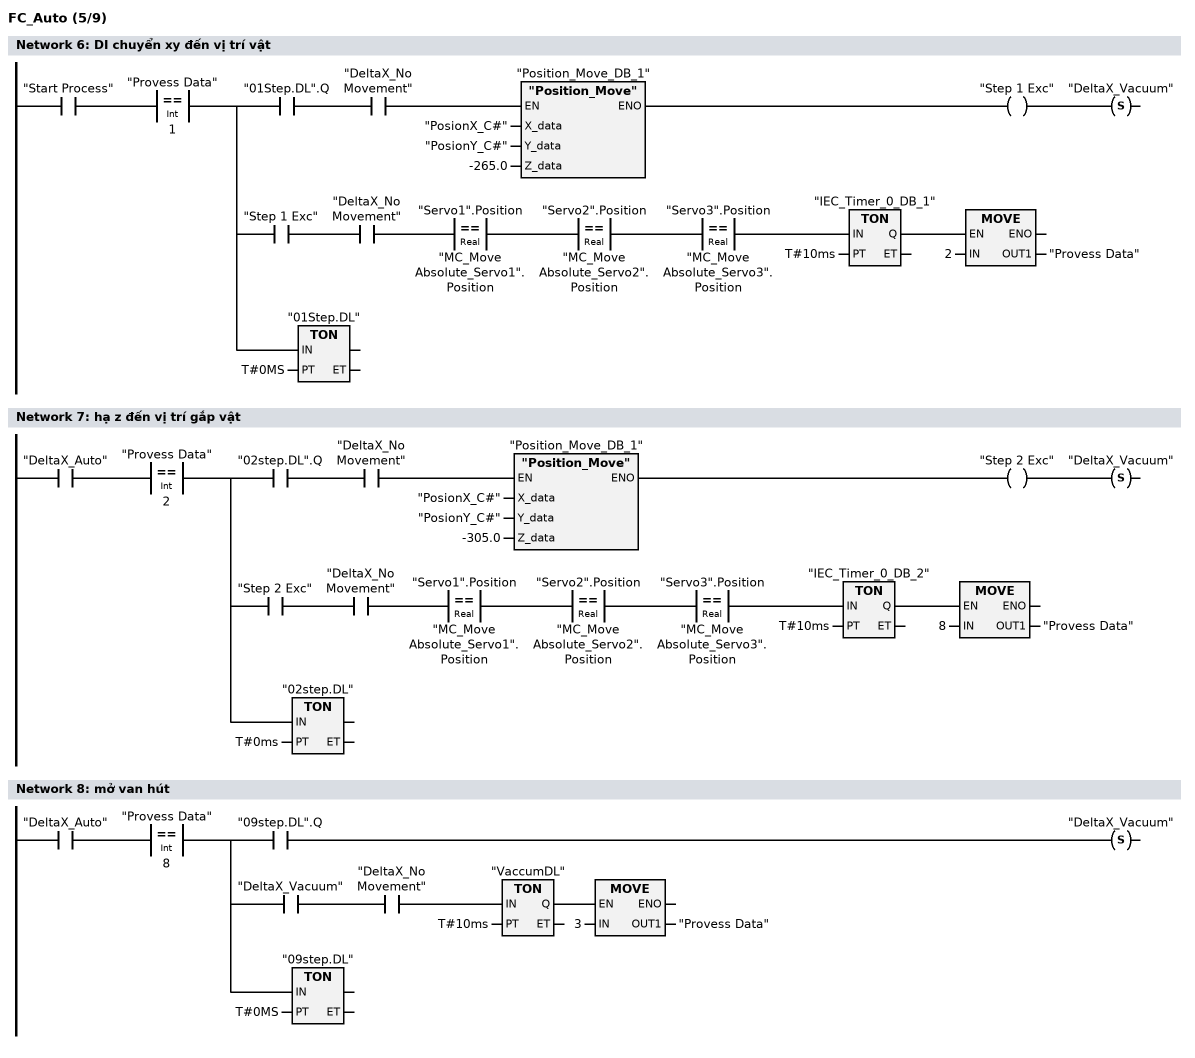
   #_w1 := "Start Process" AND ("Provess Data" = 1);
   "Position_Move_DB_1"(EN := #_w1 AND "01Step.DL".Q AND "DeltaX_No Movement",   // "Position_Move"
                        X_data := "PosionX_C#",
                        Y_data := "PosionY_C#",
                        Z_data := -265.0,
                        ENO => #_w2);
   "Step 1 Exc" := #_w2;
   IF #_w2 THEN "DeltaX_Vacuum" := TRUE; END_IF;
   "IEC_Timer_0_DB_1".TON(IN := #_w1 AND "Step 1 Exc" AND "DeltaX_No Movement" AND ("Servo1".Position = "MC_MoveAbsolute_Servo1".Position) AND ("Servo2".Position = "MC_MoveAbsolute_Servo2".Position) AND ("Servo3".Position = "MC_MoveAbsolute_Servo3".Position),
                          PT := T#10ms);
   IF "IEC_Timer_0_DB_1".Q THEN "Provess Data" := 2; END_IF;
   "01Step.DL".TON(IN := #_w1, PT := T#0MS);
END_REGION

REGION Network 7: hạ z đến vị trí gắp vật
   #_w1 := "DeltaX_Auto" AND ("Provess Data" = 2);
   "Position_Move_DB_1"(EN := #_w1 AND "02step.DL".Q AND "DeltaX_No Movement",   // "Position_Move"
                        X_data := "PosionX_C#",
                        Y_data := "PosionY_C#",
                        Z_data := -305.0,
                        ENO => #_w2);
   "Step 2 Exc" := #_w2;
   IF #_w2 THEN "DeltaX_Vacuum" := TRUE; END_IF;
   "IEC_Timer_0_DB_2".TON(IN := #_w1 AND "Step 2 Exc" AND "DeltaX_No Movement" AND ("Servo1".Position = "MC_MoveAbsolute_Servo1".Position) AND ("Servo2".Position = "MC_MoveAbsolute_Servo2".Position) AND ("Servo3".Position = "MC_MoveAbsolute_Servo3".Position),
                          PT := T#10ms);
   IF "IEC_Timer_0_DB_2".Q THEN "Provess Data" := 8; END_IF;
   "02step.DL".TON(IN := #_w1, PT := T#0ms);
END_REGION

REGION Network 8: mở van hút
   #_w1 := "DeltaX_Auto" AND ("Provess Data" = 8);
   IF #_w1 AND "09step.DL".Q THEN "DeltaX_Vacuum" := TRUE; END_IF;
   "VaccumDL".TON(IN := #_w1 AND "DeltaX_Vacuum" AND "DeltaX_No Movement", PT := T#10ms);
   IF "VaccumDL".Q THEN "Provess Data" := 3; END_IF;
   "09step.DL".TON(IN := #_w1, PT := T#0MS);
END_REGION

REGION Network 9: di chuyển z lên
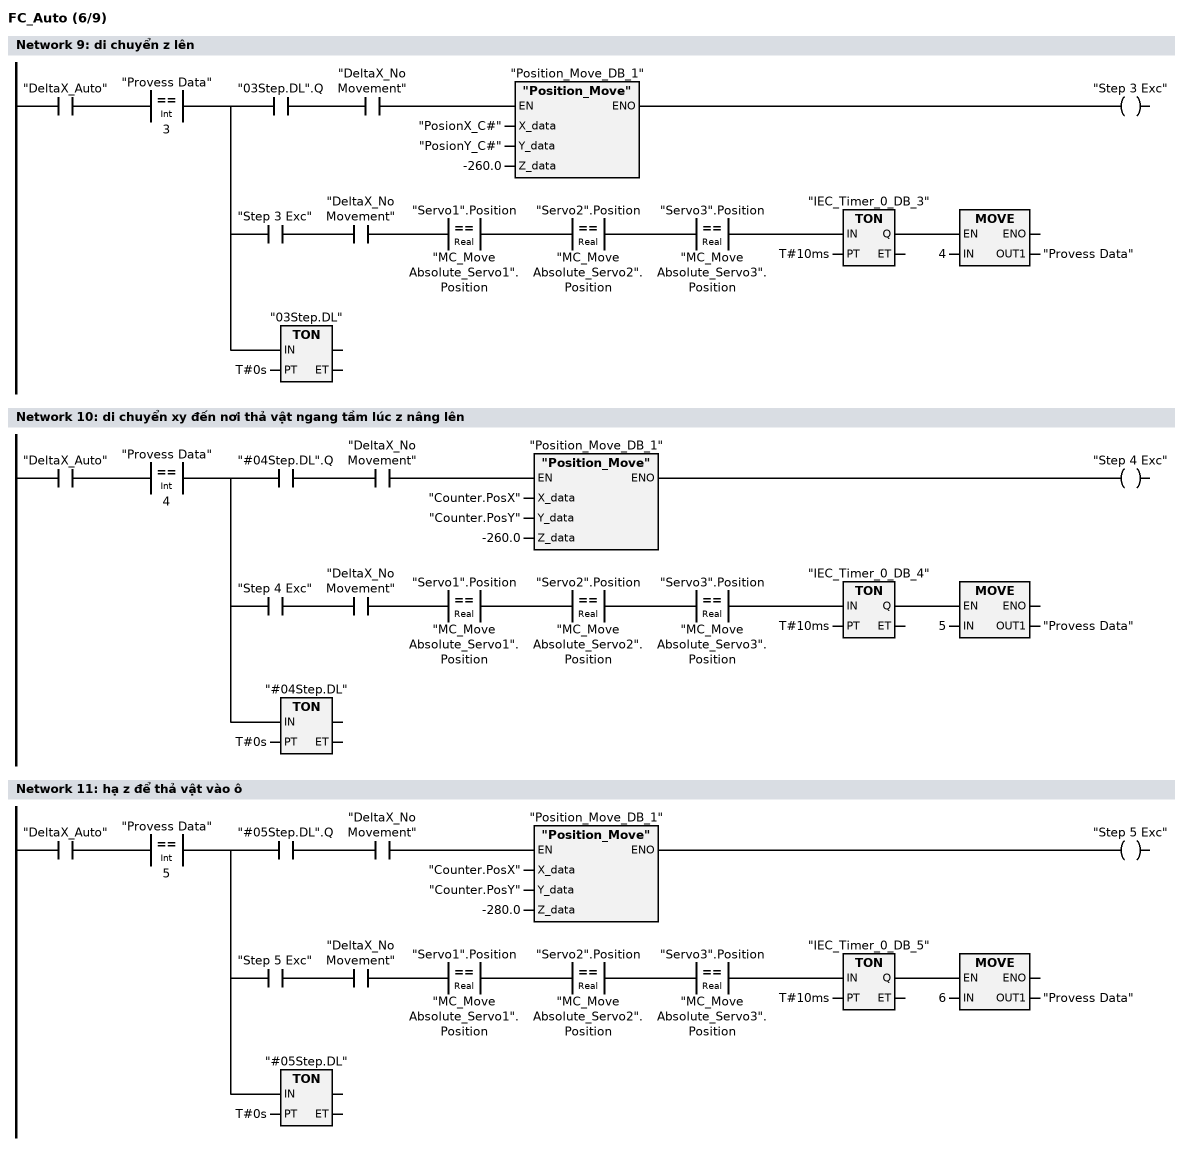
   #_w1 := "DeltaX_Auto" AND ("Provess Data" = 3);
   "Position_Move_DB_1"(EN := #_w1 AND "03Step.DL".Q AND "DeltaX_No Movement",   // "Position_Move"
                        X_data := "PosionX_C#",
                        Y_data := "PosionY_C#",
                        Z_data := -260.0,
                        ENO => #_w2);
   "Step 3 Exc" := #_w2;
   "IEC_Timer_0_DB_3".TON(IN := #_w1 AND "Step 3 Exc" AND "DeltaX_No Movement" AND ("Servo1".Position = "MC_MoveAbsolute_Servo1".Position) AND ("Servo2".Position = "MC_MoveAbsolute_Servo2".Position) AND ("Servo3".Position = "MC_MoveAbsolute_Servo3".Position),
                          PT := T#10ms);
   IF "IEC_Timer_0_DB_3".Q THEN "Provess Data" := 4; END_IF;
   "03Step.DL".TON(IN := #_w1, PT := T#0s);
END_REGION

REGION Network 10: di chuyển xy đến nơi thả vật ngang tầm lúc z nâng lên
   #_w1 := "DeltaX_Auto" AND ("Provess Data" = 4);
   "Position_Move_DB_1"(EN := #_w1 AND "#04Step.DL".Q AND "DeltaX_No Movement",   // "Position_Move"
                        X_data := "Counter.PosX",
                        Y_data := "Counter.PosY",
                        Z_data := -260.0,
                        ENO => #_w2);
   "Step 4 Exc" := #_w2;
   "IEC_Timer_0_DB_4".TON(IN := #_w1 AND "Step 4 Exc" AND "DeltaX_No Movement" AND ("Servo1".Position = "MC_MoveAbsolute_Servo1".Position) AND ("Servo2".Position = "MC_MoveAbsolute_Servo2".Position) AND ("Servo3".Position = "MC_MoveAbsolute_Servo3".Position),
                          PT := T#10ms);
   IF "IEC_Timer_0_DB_4".Q THEN "Provess Data" := 5; END_IF;
   "#04Step.DL".TON(IN := #_w1, PT := T#0s);
END_REGION

REGION Network 11: hạ z để thả vật vào ô
   #_w1 := "DeltaX_Auto" AND ("Provess Data" = 5);
   "Position_Move_DB_1"(EN := #_w1 AND "#05Step.DL".Q AND "DeltaX_No Movement",   // "Position_Move"
                        X_data := "Counter.PosX",
                        Y_data := "Counter.PosY",
                        Z_data := -280.0,
                        ENO => #_w2);
   "Step 5 Exc" := #_w2;
   "IEC_Timer_0_DB_5".TON(IN := #_w1 AND "Step 5 Exc" AND "DeltaX_No Movement" AND ("Servo1".Position = "MC_MoveAbsolute_Servo1".Position) AND ("Servo2".Position = "MC_MoveAbsolute_Servo2".Position) AND ("Servo3".Position = "MC_MoveAbsolute_Servo3".Position),
                          PT := T#10ms);
   IF "IEC_Timer_0_DB_5".Q THEN "Provess Data" := 6; END_IF;
   "#05Step.DL".TON(IN := #_w1, PT := T#0s);
END_REGION

REGION Network 12: nâng z lên lại để về vị trí ss
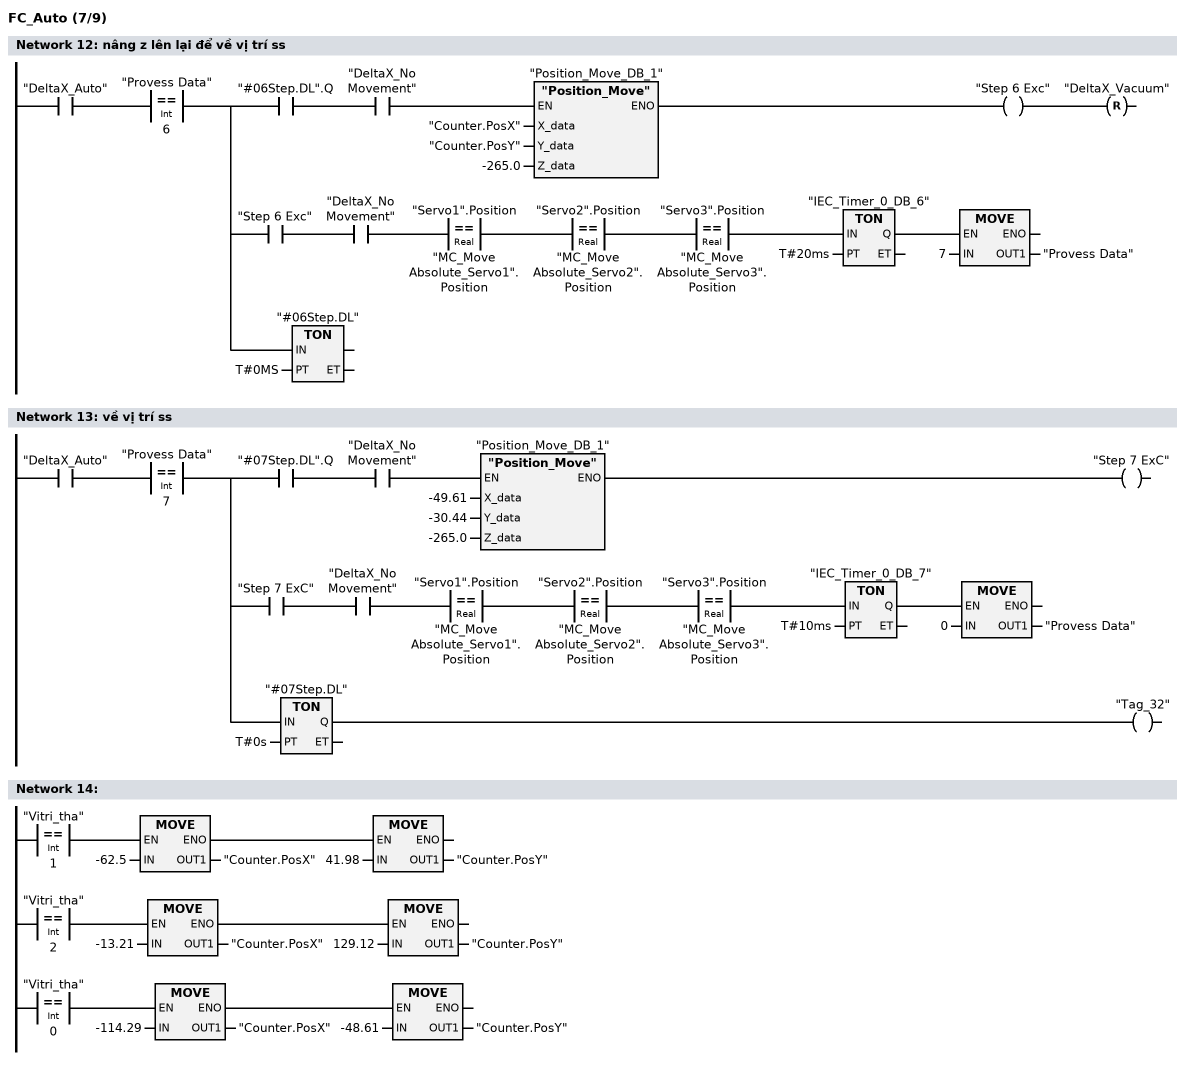
   #_w1 := "DeltaX_Auto" AND ("Provess Data" = 6);
   "Position_Move_DB_1"(EN := #_w1 AND "#06Step.DL".Q AND "DeltaX_No Movement",   // "Position_Move"
                        X_data := "Counter.PosX",
                        Y_data := "Counter.PosY",
                        Z_data := -265.0,
                        ENO => #_w2);
   "Step 6 Exc" := #_w2;
   IF #_w2 THEN "DeltaX_Vacuum" := FALSE; END_IF;
   "IEC_Timer_0_DB_6".TON(IN := #_w1 AND "Step 6 Exc" AND "DeltaX_No Movement" AND ("Servo1".Position = "MC_MoveAbsolute_Servo1".Position) AND ("Servo2".Position = "MC_MoveAbsolute_Servo2".Position) AND ("Servo3".Position = "MC_MoveAbsolute_Servo3".Position),
                          PT := T#20ms);
   IF "IEC_Timer_0_DB_6".Q THEN "Provess Data" := 7; END_IF;
   "#06Step.DL".TON(IN := #_w1, PT := T#0MS);
END_REGION

REGION Network 13: về vị trí ss
   #_w1 := "DeltaX_Auto" AND ("Provess Data" = 7);
   "Position_Move_DB_1"(EN := #_w1 AND "#07Step.DL".Q AND "DeltaX_No Movement",   // "Position_Move"
                        X_data := -49.61,
                        Y_data := -30.44,
                        Z_data := -265.0,
                        ENO => #_w2);
   "Step 7 ExC" := #_w2;
   "IEC_Timer_0_DB_7".TON(IN := #_w1 AND "Step 7 ExC" AND "DeltaX_No Movement" AND ("Servo1".Position = "MC_MoveAbsolute_Servo1".Position) AND ("Servo2".Position = "MC_MoveAbsolute_Servo2".Position) AND ("Servo3".Position = "MC_MoveAbsolute_Servo3".Position),
                          PT := T#10ms);
   IF "IEC_Timer_0_DB_7".Q THEN "Provess Data" := 0; END_IF;
   "#07Step.DL".TON(IN := #_w1, PT := T#0s);
   "Tag_32" := "#07Step.DL".Q;
END_REGION

REGION Network 14
   RUNG wire#powerrail
      { S7_Templates := "SrcType := Int" } EQ_Contact(in1 := "Vitri_tha", in2 := 1)
      Move(in := -62.5, out1 => "Counter.PosX")
      Move(in := 41.98, out1 => "Counter.PosY")
   END_RUNG
   RUNG wire#powerrail
      { S7_Templates := "SrcType := Int" } EQ_Contact(in1 := "Vitri_tha", in2 := 2)
      Move(in := -13.21, out1 => "Counter.PosX")
      Move(in := 129.12, out1 => "Counter.PosY")
   END_RUNG
   RUNG wire#powerrail
      { S7_Templates := "SrcType := Int" } EQ_Contact(in1 := "Vitri_tha", in2 := 0)
      Move(in := -114.29, out1 => "Counter.PosX")
      Move(in := -48.61, out1 => "Counter.PosY")
   END_RUNG
   // the same network as SCL:
   IF "Vitri_tha" = 1 THEN
       "Counter.PosX" := -62.5;
       "Counter.PosY" := 41.98;
   END_IF;
   IF "Vitri_tha" = 2 THEN
       "Counter.PosX" := -13.21;
       "Counter.PosY" := 129.12;
   END_IF;
   IF "Vitri_tha" = 0 THEN
       "Counter.PosX" := -114.29;
       "Counter.PosY" := -48.61;
   END_IF;
END_REGION

REGION Network 15
